KUKA KRL program: MyProgram_063().src

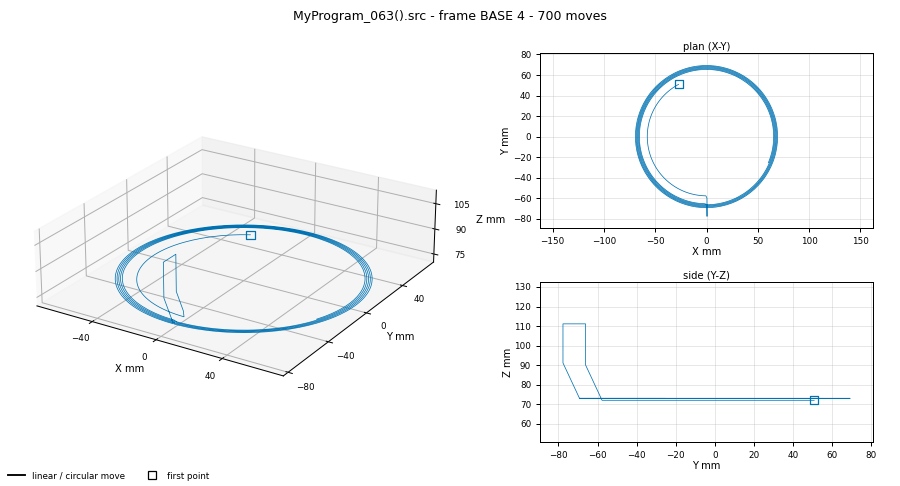
[picture p0: tool path of MyProgram_063().src in frame BASE 4, 700 of 700 moves have a stored position in this frame; points joined in program order, loops and branches not executed]
&ACCESS RVP
&REL 1
&PARAM TEMPLATE = C:\KRC\Roboter\Template\vorgabe
&PARAM EDITMASK = *
DEF MyProgram_063()
; ---- Setting reference (Base) ----
$BASE = BASE_DATA[4]

; --------------------------
; ---- Setting tool (TCP) ----
$TOOL = TOOL_DATA[3]
; --------------------------

$VEL.CP = VEL_APROX_PRINT
Startdeposition()
$VEL.CP = VEL_PRINT
LIN {X -27.2088,Y 50.891,Z 72,A 112.2891,B 24.8573,C -2.7565,E1 24.923,E2 -28.5413} C_DIS
LIN {X -29.6669,Y 49.4984,Z 72,A 115.1236,B 24.8577,C -2.7521,E1 24.9161,E2 -31.3738} C_DIS
LIN {X -32.0537,Y 47.9875,Z 72,A 117.9461,B 24.8583,C -2.7472,E1 24.9095,E2 -34.1937} C_DIS
LIN {X -34.3644,Y 46.3604,Z 72,A 120.7752,B 24.8588,C -2.742,E1 24.9031,E2 -37.0202} C_DIS
LIN {X -36.6119,Y 44.6068,Z 72,A 123.5826,B 24.8595,C -2.7356,E1 24.897,E2 -39.8228} C_DIS
LIN {X -38.7479,Y 42.7649,Z 72,A 126.4499,B 24.86,C -2.7305,E1 24.891,E2 -42.6893} C_DIS
LIN {X -40.7899,Y 40.8218,Z 72,A 129.2609,B 24.8606,C -2.7241,E1 24.8854,E2 -45.4969} C_DIS
LIN {X -42.7465,Y 38.7683,Z 72,A 132.0709,B 24.8613,C -2.7171,E1 24.8801,E2 -48.3025} C_DIS
LIN {X -44.6073,Y 36.6114,Z 72,A 134.9183,B 24.862,C -2.7103,E1 24.875,E2 -51.1466} C_DIS
LIN {X -46.3432,Y 34.3876,Z 72,A 137.7118,B 24.8628,C -2.7028,E1 24.8703,E2 -53.9356} C_DIS
LIN {X -47.9666,Y 32.0848,Z 72,A 140.5939,B 24.8634,C -2.6967,E1 24.8657,E2 -56.8174} C_DIS
LIN {X -49.5558,Y 29.5705,Z 72,A 143.4336,B 24.8645,C -2.6865,E1 24.8616,E2 -59.6473} C_DIS
LIN {X -50.8913,Y 27.2082,Z 72,A 146.2802,B 24.865,C -2.6814,E1 24.8578,E2 -62.4967} C_DIS
LIN {X -52.2094,Y 24.5834,Z 72,A 149.1598,B 24.8659,C -2.6723,E1 24.8543,E2 -65.37} C_DIS
LIN {X -53.3151,Y 22.0828,Z 72,A 151.9081,B 24.8667,C -2.6647,E1 24.8512,E2 -68.1155} C_DIS
LIN {X -54.3384,Y 19.4281,Z 72,A 154.7769,B 24.8674,C -2.657,E1 24.8485,E2 -70.9819} C_DIS
LIN {X -55.2245,Y 16.7453,Z 72,A 157.5583,B 24.8683,C -2.6479,E1 24.8461,E2 -73.7577} C_DIS
LIN {X -56.0051,Y 13.9133,Z 72,A 160.45,B 24.8693,C -2.6385,E1 24.8441,E2 -76.6436} C_DIS
LIN {X -56.5972,Y 11.2653,Z 72,A 163.2006,B 24.87,C -2.631,E1 24.8425,E2 -79.3926} C_DIS
LIN {X -57.0834,Y 8.4678,Z 72,A 166.0768,B 24.8708,C -2.6231,E1 24.8412,E2 -82.2669} C_DIS
LIN {X -57.43,Y 5.6498,Z 72,A 168.848,B 24.8718,C -2.6134,E1 24.8404,E2 -85.0315} C_DIS
LIN {X -57.638,Y 2.8318,Z 72,A 171.7312,B 24.8725,C -2.6058,E1 24.8399,E2 -87.914} C_DIS
LIN {X -57.7082,Y -0.0206,Z 72,A 174.6003,B 24.8733,C -2.5975,E1 24.8398,E2 -90.7805} C_DIS
LIN {X -57.6375,Y -2.8407,Z 72,A 177.3607,B 24.8742,C -2.588,E1 24.8401,E2 -93.5348} C_DIS
LIN {X -57.4183,Y -5.7684,Z 72,A -179.6933,B 24.8751,C -2.5795,E1 24.8408,E2 -96.478} C_DIS
LIN {X -57.0846,Y -8.4591,Z 72,A -176.9668,B 24.8758,C -2.5717,E1 24.8418,E2 -99.2022} C_DIS
LIN {X -56.5987,Y -11.258,Z 72,A -174.1104,B 24.8766,C -2.5637,E1 24.8433,E2 -102.0565} C_DIS
LIN {X -55.9773,Y -14.0247,Z 72,A -171.2895,B 24.8774,C -2.5553,E1 24.8451,E2 -104.8738} C_DIS
LIN {X -55.2229,Y -16.7506,Z 72,A -168.4174,B 24.8781,C -2.548,E1 24.8473,E2 -107.7451} C_DIS
LIN {X -54.3355,Y -19.4363,Z 72,A -165.6279,B 24.8789,C -2.5396,E1 24.8499,E2 -110.5302} C_DIS
LIN {X -53.3047,Y -22.108,Z 72,A -162.771,B 24.8797,C -2.5317,E1 24.8528,E2 -113.3843} C_DIS
LIN {X -52.1127,Y -24.7874,Z 72,A -159.8924,B 24.8805,C -2.523,E1 24.8562,E2 -116.2579} C_DIS
LIN {X -50.8921,Y -27.2066,Z 72,A -157.1453,B 24.8811,C -2.5168,E1 24.8597,E2 -119.0047} C_DIS
LIN {X -49.5012,Y -29.6623,Z 72,A -154.3076,B 24.8817,C -2.51,E1 24.8637,E2 -121.8411} C_DIS
LIN {X -47.9927,Y -32.0459,Z 72,A -151.4699,B 24.8823,C -2.5036,E1 24.868,E2 -124.6778} C_DIS
LIN {X -46.3598,Y -34.3651,Z 72,A -148.6733,B 24.883,C -2.4965,E1 24.8726,E2 -127.4709} C_DIS
LIN {X -44.6722,Y -36.5319,Z 72,A -145.9581,B 24.8836,C -2.4899,E1 24.8773,E2 -130.1831} C_DIS
LIN {X -42.9715,Y -38.5173,Z 72,A -143.3305,B 24.8841,C -2.4847,E1 24.8822,E2 -132.8102} C_DIS
LIN {X -41.017,Y -40.5923,Z 72,A -140.4968,B 24.8847,C -2.4788,E1 24.8877,E2 -135.642} C_DIS
LIN {X -38.9797,Y -42.5525,Z 72,A -137.6509,B 24.8851,C -2.4739,E1 24.8935,E2 -138.4878} C_DIS
LIN {X -36.8321,Y -44.4244,Z 72,A -134.8917,B 24.8857,C -2.4673,E1 24.8993,E2 -141.2419} C_DIS
LIN {X -34.7623,Y -46.0622,Z 72,A -132.2373,B 24.8861,C -2.4633,E1 24.9052,E2 -143.8966} C_DIS
LIN {X -32.6406,Y -47.5903,Z 72,A -129.5668,B 24.8864,C -2.4605,E1 24.9113,E2 -146.5694} C_DIS
LIN {X -30.2771,Y -49.1274,Z 72,A -126.7787,B 24.8868,C -2.4561,E1 24.9179,E2 -149.356} C_DIS
LIN {X -27.8422,Y -50.5472,Z 72,A -123.9046,B 24.887,C -2.4537,E1 24.9249,E2 -152.2328} C_DIS
LIN {X -25.3395,Y -51.8463,Z 72,A -121.1321,B 24.8874,C -2.4498,E1 24.9318,E2 -155.0034} C_DIS
LIN {X -22.7304,Y -53.0422,Z 72,A -118.294,B 24.8877,C -2.4465,E1 24.939,E2 -157.8405} C_DIS
LIN {X -19.9996,Y -54.1309,Z 72,A -115.4113,B 24.888,C -2.4431,E1 24.9465,E2 -160.7212} C_DIS
LIN {X -17.431,Y -55.0116,Z 72,A -112.6658,B 24.888,C -2.442,E1 24.9538,E2 -163.4692} C_DIS
LIN {X -14.707,Y -55.8019,Z 72,A -109.8374,B 24.8882,C -2.4405,E1 24.9614,E2 -166.2983} C_DIS
LIN {X -11.8501,Y -56.478,Z 72,A -106.9721,B 24.8884,C -2.4382,E1 24.9692,E2 -169.1617} C_DIS
LIN {X -9.1675,Y -56.9755,Z 72,A -104.197,B 24.8884,C -2.4386,E1 24.9769,E2 -171.9406} C_DIS
LIN {X -6.3785,Y -57.3539,Z 72,A -101.389,B 24.8884,C -2.4385,E1 24.9847,E2 -174.7502} C_DIS
LIN {X -3.4748,Y -57.6033,Z 72,A -98.5125,B 24.8884,C -2.4381,E1 24.9927,E2 -177.627} C_DIS
LIN {X -0.6243,Y -57.7045,Z 72,A -95.7298,B 24.8884,C -2.4375,E1 25.0004,E2 -180.4086} C_DIS
LIN {X -0.6243,Y -57.7045,Z 72,A -95.7298,B 24.8884,C -2.4375,E1 25.0004,E2 -180.4086} C_DIS
Enddeposition()
LIN {X 0.4164,Y -59.8168,Z 76.5315,A -95.6722,B 24.8907,C -2.4133,E1 25.0004,E2 -180.4086} C_DIS
LIN {X 0.4214,Y -66.1561,Z 90.1262,A -95.6453,B 24.8917,C -2.402,E1 25.0004,E2 -180.4086} C_DIS
LIN {X 0.4214,Y -66.1561,Z 111.1262,A -96.001,B 24.8778,C -2.5516,E1 25.0004,E2 -180.4086} C_DIS
LIN {X 0.5054,Y -77.7039,Z 111.1262,A -95.259,B 24.8948,C -2.368,E1 25.0013,E2 -180.7142} C_DIS
LIN {X 0.5054,Y -77.7039,Z 91.1262,A -94.9205,B 24.9071,C -2.2255,E1 25.0013,E2 -180.7142} C_DIS
LIN {X 0.4665,Y -71.3647,Z 77.5315,A -94.9453,B 24.9062,C -2.2359,E1 25.0013,E2 -180.7142} C_DIS
LIN {X 0.4536,Y -69.2517,Z 73,A -94.9551,B 24.9059,C -2.2401,E1 25.0013,E2 -180.7142} C_DIS
Startdeposition()
$VEL.CP = VEL_PRINT
LIN {X -1.6996,Y -69.2353,Z 73,A -97.3478,B 24.9072,C -2.2246,E1 24.9945,E2 -178.2848} C_DIS
LIN {X -4.2468,Y -69.1258,Z 73,A -99.457,B 24.9072,C -2.2246,E1 24.9886,E2 -176.1746} C_DIS
LIN {X -6.7883,Y -68.9227,Z 73,A -101.3578,B 24.9067,C -2.2297,E1 24.9834,E2 -174.2852} C_DIS
LIN {X -9.3205,Y -68.6261,Z 73,A -103.6767,B 24.9071,C -2.225,E1 24.9769,E2 -171.9535} C_DIS
LIN {X -11.9777,Y -68.2118,Z 73,A -105.8535,B 24.907,C -2.2268,E1 24.9709,E2 -169.7789} C_DIS
LIN {X -15.0376,Y -67.6032,Z 73,A -108.2937,B 24.9066,C -2.2313,E1 24.9643,E2 -167.3464} C_DIS
LIN {X -17.651,Y -66.9691,Z 73,A -110.7147,B 24.9069,C -2.2278,E1 24.9577,E2 -164.9138} C_DIS
LIN {X -20.104,Y -66.274,Z 73,A -112.8273,B 24.9068,C -2.2292,E1 24.952,E2 -162.8009} C_DIS
LIN {X -22.5297,Y -65.4891,Z 73,A -114.914,B 24.9066,C -2.2314,E1 24.9465,E2 -160.7155} C_DIS
LIN {X -24.9249,Y -64.6155,Z 73,A -116.8452,B 24.9061,C -2.2374,E1 24.9415,E2 -158.7948} C_DIS
LIN {X -27.2864,Y -63.6543,Z 73,A -119.1684,B 24.9063,C -2.2346,E1 24.9355,E2 -156.4595} C_DIS
LIN {X -29.6108,Y -62.6068,Z 73,A -121.2832,B 24.9061,C -2.2368,E1 24.9301,E2 -154.3447} C_DIS
LIN {X -31.8951,Y -61.4745,Z 73,A -123.3985,B 24.9059,C -2.2393,E1 24.9249,E2 -152.2297} C_DIS
LIN {X -34.2574,Y -60.1892,Z 73,A -125.5804,B 24.9056,C -2.2433,E1 24.9195,E2 -150.051} C_DIS
LIN {X -36.9333,Y -58.5854,Z 73,A -127.9318,B 24.9048,C -2.2523,E1 24.914,E2 -147.7136} C_DIS
LIN {X -38.5924,Y -57.506,Z 73,A -129.8132,B 24.9051,C -2.2493,E1 24.9096,E2 -145.819} C_DIS
LIN {X -41.1431,Y -55.7096,Z 73,A -132.1658,B 24.9043,C -2.2588,E1 24.9043,E2 -143.4807} C_DIS
LIN {X -43.1657,Y -54.1575,Z 73,A -134.2837,B 24.904,C -2.2623,E1 24.8996,E2 -141.3635} C_DIS
LIN {X -45.0032,Y -52.6399,Z 73,A -136.5418,B 24.9042,C -2.2596,E1 24.8947,E2 -139.0901} C_DIS
LIN {X -47.2376,Y -50.6451,Z 73,A -138.9913,B 24.9037,C -2.2651,E1 24.8897,E2 -136.6439} C_DIS
LIN {X -49.4705,Y -48.4663,Z 73,A -141.3461,B 24.9029,C -2.2754,E1 24.885,E2 -134.3039} C_DIS
LIN {X -51.2209,Y -46.6126,Z 73,A -143.5601,B 24.9027,C -2.2777,E1 24.8808,E2 -132.0856} C_DIS
LIN {X -52.9925,Y -44.5893,Z 73,A -145.9907,B 24.9027,C -2.2782,E1 24.8764,E2 -129.6451} C_DIS
LIN {X -54.5978,Y -42.6086,Z 73,A -148.0451,B 24.9021,C -2.2843,E1 24.8728,E2 -127.5957} C_DIS
LIN {X -56.2103,Y -40.4563,Z 73,A -150.2985,B 24.9017,C -2.2891,E1 24.8691,E2 -125.3428} C_DIS
LIN {X -57.9753,Y -37.8838,Z 73,A -152.6554,B 24.9007,C -2.3004,E1 24.8655,E2 -123.0012} C_DIS
LIN {X -59.2789,Y -35.8089,Z 73,A -154.7202,B 24.9003,C -2.3048,E1 24.8624,E2 -120.9363} C_DIS
LIN {X -60.327,Y -34.0142,Z 73,A -156.6632,B 24.9003,C -2.3046,E1 24.8597,E2 -118.9825} C_DIS
LIN {X -61.7977,Y -31.2628,Z 73,A -159.0212,B 24.8993,C -2.3163,E1 24.8567,E2 -116.64} C_DIS
LIN {X -62.883,Y -29.0176,Z 73,A -161.2043,B 24.8991,C -2.3195,E1 24.8541,E2 -114.4526} C_DIS
LIN {X -63.9843,Y -26.5032,Z 73,A -163.6722,B 24.8989,C -2.3217,E1 24.8513,E2 -111.9764} C_DIS
LIN {X -64.9644,Y -23.9988,Z 73,A -165.8612,B 24.8982,C -2.3289,E1 24.8492,E2 -109.7922} C_DIS
LIN {X -65.8037,Y -21.5914,Z 73,A -167.985,B 24.8977,C -2.3347,E1 24.8473,E2 -107.6703} C_DIS
LIN {X -66.5538,Y -19.1547,Z 73,A -170.1085,B 24.8972,C -2.3407,E1 24.8456,E2 -105.5487} C_DIS
LIN {X -67.3489,Y -16.138,Z 73,A -172.468,B 24.8961,C -2.3531,E1 24.844,E2 -103.2052} C_DIS
LIN {X -67.8973,Y -13.6481,Z 73,A -174.592,B 24.8956,C -2.3593,E1 24.8427,E2 -101.0833} C_DIS
LIN {X -68.3252,Y -11.31,Z 73,A -176.8369,B 24.8956,C -2.3595,E1 24.8417,E2 -98.8256} C_DIS
LIN {X -68.7353,Y -8.4777,Z 73,A -179.0356,B 24.8946,C -2.3704,E1 24.8408,E2 -96.6397} C_DIS
LIN {X -69.0008,Y -5.942,Z 73,A 178.6296,B 24.8944,C -2.3722,E1 24.8402,E2 -94.2955} C_DIS
LIN {X -69.1727,Y -3.3982,Z 73,A 176.5051,B 24.8938,C -2.3786,E1 24.8399,E2 -92.1733} C_DIS
LIN {X -69.2526,Y -0.6533,Z 73,A 174.2028,B 24.8932,C -2.3851,E1 24.8398,E2 -89.8728} C_DIS
LIN {X -69.2092,Y 2.5491,Z 73,A 171.5482,B 24.8925,C -2.3934,E1 24.84,E2 -87.222} C_DIS
LIN {X -69.0685,Y 5.0948,Z 73,A 169.6341,B 24.8915,C -2.4041,E1 24.8403,E2 -85.3221} C_DIS
LIN {X -68.8342,Y 7.6336,Z 73,A 167.2992,B 24.8914,C -2.4061,E1 24.841,E2 -82.9779} C_DIS
LIN {X -68.5066,Y 10.162,Z 73,A 165.1746,B 24.8908,C -2.4125,E1 24.8418,E2 -80.8558} C_DIS
LIN {X -67.9862,Y 13.1957,Z 73,A 162.8452,B 24.8896,C -2.425,E1 24.8429,E2 -78.5425} C_DIS
LIN {X -67.5419,Y 15.3103,Z 73,A 160.862,B 24.8895,C -2.4266,E1 24.8441,E2 -76.5513} C_DIS
LIN {X -66.9326,Y 17.7859,Z 73,A 158.7356,B 24.8889,C -2.4328,E1 24.8456,E2 -74.4273} C_DIS
LIN {X -66.0637,Y 20.7823,Z 73,A 156.3753,B 24.8878,C -2.4453,E1 24.8475,E2 -72.0835} C_DIS
LIN {X -65.254,Y 23.1998,Z 73,A 154.1569,B 24.8874,C -2.4495,E1 24.8495,E2 -69.8625} C_DIS
LIN {X -64.3048,Y 25.716,Z 73,A 151.7219,B 24.8872,C -2.4518,E1 24.852,E2 -67.4193} C_DIS
LIN {X -63.3146,Y 28.0655,Z 73,A 149.8086,B 24.8862,C -2.4622,E1 24.8541,E2 -65.5202} C_DIS
LIN {X -62.2387,Y 30.3769,Z 73,A 147.685,B 24.8857,C -2.4681,E1 24.8566,E2 -63.3993} C_DIS
LIN {X -61.0785,Y 32.6471,Z 73,A 145.3517,B 24.8855,C -2.4695,E1 24.8597,E2 -61.0568} C_DIS
LIN {X -59.8354,Y 34.8731,Z 73,A 143.4389,B 24.8846,C -2.4797,E1 24.8623,E2 -59.1583} C_DIS
LIN {X -58.5113,Y 37.0519,Z 73,A 141.106,B 24.8845,C -2.4808,E1 24.8657,E2 -56.8163} C_DIS
LIN {X -57.1079,Y 39.1804,Z 73,A 139.0516,B 24.8838,C -2.4878,E1 24.8689,E2 -54.7682} C_DIS
LIN {X -55.6271,Y 41.2558,Z 73,A 136.8615,B 24.8835,C -2.4917,E1 24.8725,E2 -52.5768} C_DIS
LIN {X -53.9829,Y 43.3839,Z 73,A 134.6734,B 24.8828,C -2.4983,E1 24.8763,E2 -50.3942} C_DIS
LIN {X -51.9742,Y 45.7711,Z 73,A 132.222,B 24.882,C -2.5076,E1 24.8807,E2 -47.9538} C_DIS
LIN {X -50.1586,Y 47.7549,Z 73,A 130.0004,B 24.8815,C -2.5131,E1 24.885,E2 -45.7355} C_DIS
LIN {X -48.3669,Y 49.5688,Z 73,A 127.6695,B 24.8815,C -2.5133,E1 24.8896,E2 -43.3954} C_DIS
LIN {X -46.5096,Y 51.3154,Z 73,A 125.5493,B 24.881,C -2.5179,E1 24.894,E2 -41.2775} C_DIS
LIN {X -44.4818,Y 53.0819,Z 73,A 123.3632,B 24.8805,C -2.5236,E1 24.8986,E2 -39.0966} C_DIS
LIN {X -42.0461,Y 55.0313,Z 73,A 121.0085,B 24.8795,C -2.534,E1 24.9037,E2 -36.758} C_DIS
LIN {X -39.992,Y 56.5416,Z 73,A 118.8893,B 24.8791,C -2.538,E1 24.9085,E2 -34.641} C_DIS
LIN {X -37.8838,Y 57.9753,Z 73,A 116.6766,B 24.8789,C -2.5398,E1 24.9136,E2 -32.4252} C_DIS
LIN {X -35.6048,Y 59.403,Z 73,A 114.2482,B 24.8789,C -2.5394,E1 24.9194,E2 -29.9882} C_DIS
LIN {X -33.3942,Y 60.6732,Z 73,A 112.3403,B 24.8782,C -2.5474,E1 24.9241,E2 -28.094} C_DIS
LIN {X -31.1384,Y 61.8613,Z 73,A 110.0136,B 24.8783,C -2.546,E1 24.9299,E2 -25.7576} C_DIS
LIN {X -28.7129,Y 63.0229,Z 73,A 107.8309,B 24.8779,C -2.5503,E1 24.9354,E2 -23.5797} C_DIS
LIN {X -25.8454,Y 64.2521,Z 73,A 105.3814,B 24.8773,C -2.5569,E1 24.9417,E2 -21.1403} C_DIS
LIN {X -23.3317,Y 65.2077,Z 73,A 102.9603,B 24.8774,C -2.5553,E1 24.948,E2 -18.7105} C_DIS
LIN {X -20.7823,Y 66.0637,Z 73,A 100.7794,B 24.8771,C -2.5589,E1 24.9538,E2 -16.5341} C_DIS
LIN {X -17.7859,Y 66.9326,Z 73,A 98.2119,B 24.8768,C -2.5619,E1 24.9607,E2 -13.9697} C_DIS
LIN {X -15.0376,Y 67.6032,Z 73,A 95.8468,B 24.8766,C -2.5634,E1 24.9671,E2 -11.6051} C_DIS
LIN {X -11.9777,Y 68.2118,Z 73,A 93.2608,B 24.8765,C -2.5653,E1 24.9742,E2 -9.0209} C_DIS
LIN {X -9.1819,Y 68.6441,Z 73,A 90.9169,B 24.8763,C -2.5667,E1 24.9807,E2 -6.6784} C_DIS
LIN {X -6.0812,Y 68.9879,Z 73,A 88.5704,B 24.8757,C -2.5736,E1 24.9872,E2 -4.3469} C_DIS
LIN {X -4.1073,Y 69.1335,Z 73,A 86.6937,B 24.8761,C -2.5686,E1 24.9924,E2 -2.4576} C_DIS
LIN {X -0.9896,Y 69.2484,Z 73,A 84.2546,B 24.8757,C -2.5727,E1 24.9992,E2 -0.028} C_DIS
LIN {X 1.6996,Y 69.2353,Z 73,A 81.8355,B 24.8762,C -2.5684,E1 25.006,E2 2.401} C_DIS
LIN {X 4.2468,Y 69.1258,Z 73,A 79.7364,B 24.8762,C -2.5687,E1 25.0119,E2 4.4987} C_DIS
LIN {X 6.7883,Y 68.9227,Z 73,A 77.8259,B 24.8757,C -2.5733,E1 25.0171,E2 6.3972} C_DIS
LIN {X 9.3205,Y 68.6261,Z 73,A 75.5089,B 24.8762,C -2.5678,E1 25.0236,E2 8.7254} C_DIS
LIN {X 11.8402,Y 68.2365,Z 73,A 73.4007,B 24.8762,C -2.5671,E1 25.0294,E2 10.8329} C_DIS
LIN {X 14.3437,Y 67.7545,Z 73,A 71.5022,B 24.8759,C -2.5714,E1 25.0346,E2 12.7191} C_DIS
LIN {X 16.8279,Y 67.1806,Z 73,A 69.3955,B 24.8759,C -2.5703,E1 25.0403,E2 14.8254} C_DIS
LIN {X 19.2892,Y 66.5157,Z 73,A 67.0806,B 24.8766,C -2.5638,E1 25.0465,E2 17.1519} C_DIS
LIN {X 21.8568,Y 65.716,Z 73,A 64.9092,B 24.8766,C -2.5634,E1 25.0523,E2 19.3202} C_DIS
LIN {X 24.7942,Y 64.665,Z 73,A 62.5704,B 24.8763,C -2.5671,E1 25.0584,E2 21.6453} C_DIS
LIN {X 26.632,Y 63.9301,Z 73,A 60.6996,B 24.877,C -2.5596,E1 25.0633,E2 23.5296} C_DIS
LIN {X 29.4841,Y 62.6658,Z 73,A 58.3618,B 24.8767,C -2.5628,E1 25.0692,E2 25.8539} C_DIS
LIN {X 31.7707,Y 61.5381,Z 73,A 56.1647,B 24.8772,C -2.5579,E1 25.0747,E2 28.0566} C_DIS
LIN {X 34.1362,Y 60.2589,Z 73,A 53.962,B 24.8774,C -2.5555,E1 25.08,E2 30.2587} C_DIS
LIN {X 36.3311,Y 58.9616,Z 73,A 51.6513,B 24.8782,C -2.5472,E1 25.0856,E2 32.5817} C_DIS
LIN {X 38.4767,Y 57.5844,Z 73,A 49.797,B 24.8779,C -2.5505,E1 25.0899,E2 34.4223} C_DIS
LIN {X 40.5701,Y 56.1291,Z 73,A 47.4764,B 24.8787,C -2.5415,E1 25.0952,E2 36.756} C_DIS
LIN {X 42.6086,Y 54.5978,Z 73,A 45.3469,B 24.8792,C -2.5372,E1 25.0999,E2 38.8879} C_DIS
LIN {X 44.6957,Y 52.9019,Z 73,A 43.1809,B 24.8794,C -2.5346,E1 25.1046,E2 41.0518} C_DIS
LIN {X 47.0328,Y 50.8353,Z 73,A 40.8475,B 24.8793,C -2.536,E1 25.1094,E2 43.3725} C_DIS
LIN {X 48.4663,Y 49.4705,Z 73,A 38.9811,B 24.8802,C -2.5266,E1 25.1132,E2 45.2533} C_DIS
LIN {X 50.6451,Y 47.2376,Z 73,A 36.6485,B 24.8801,C -2.5276,E1 25.1177,E2 47.5735} C_DIS
LIN {X 52.3494,Y 45.3415,Z 73,A 34.4563,B 24.8807,C -2.5207,E1 25.1217,E2 49.7722} C_DIS
LIN {X 54.0709,Y 43.2754,Z 73,A 32.0505,B 24.8817,C -2.5108,E1 25.126,E2 52.1904} C_DIS
LIN {X 55.6271,Y 41.2558,Z 73,A 29.9525,B 24.8821,C -2.506,E1 25.1295,E2 54.2898} C_DIS
LIN {X 57.1079,Y 39.1804,Z 73,A 28.0625,B 24.8821,C -2.5066,E1 25.1325,E2 56.1691} C_DIS
LIN {X 58.5113,Y 37.0519,Z 73,A 25.7574,B 24.8831,C -2.496,E1 25.1361,E2 58.4877} C_DIS
LIN {X 59.9051,Y 34.752,Z 73,A 23.5949,B 24.8835,C -2.4918,E1 25.1391,E2 60.6489} C_DIS
LIN {X 61.1436,Y 32.5235,Z 73,A 21.4983,B 24.884,C -2.4865,E1 25.1419,E2 62.7471} C_DIS
LIN {X 62.5463,Y 29.7368,Z 73,A 19.1689,B 24.884,C -2.4862,E1 25.1448,E2 65.0648} C_DIS
LIN {X 63.5984,Y 27.4145,Z 73,A 17.0727,B 24.8845,C -2.4806,E1 25.1472,E2 67.1627} C_DIS
LIN {X 64.5644,Y 25.055,Z 73,A 14.8837,B 24.8853,C -2.4724,E1 25.1494,E2 69.359} C_DIS
LIN {X 65.4891,Y 22.5297,Z 73,A 12.6887,B 24.8858,C -2.4667,E1 25.1515,E2 71.5551} C_DIS
LIN {X 66.274,Y 20.104,Z 73,A 10.5932,B 24.8863,C -2.4609,E1 25.1533,E2 73.6526} C_DIS
LIN {X 66.9691,Y 17.651,Z 73,A 8.2903,B 24.8874,C -2.4492,E1 25.155,E2 75.9697} C_DIS
LIN {X 67.6032,Y 15.0376,Z 73,A 6.13,B 24.8879,C -2.4443,E1 25.1563,E2 78.1293} C_DIS
LIN {X 68.2118,Y 11.9777,Z 73,A 3.8022,B 24.8879,C -2.4433,E1 25.1575,E2 80.4458} C_DIS
LIN {X 68.5262,Y 10.0236,Z 73,A 1.9402,B 24.889,C -2.432,E1 25.1583,E2 82.3234} C_DIS
LIN {X 68.8487,Y 7.4946,Z 73,A -0.1544,B 24.8896,C -2.4258,E1 25.159,E2 84.4202} C_DIS
LIN {X 69.1164,Y 4.3863,Z 73,A -2.4819,B 24.8896,C -2.4247,E1 25.1595,E2 86.7366} C_DIS
LIN {X 69.231,Y 1.8393,Z 73,A -4.6824,B 24.8905,C -2.4155,E1 25.1598,E2 88.9458} C_DIS
LIN {X 69.2484,Y -0.9896,Z 73,A -7.1363,B 24.8915,C -2.405,E1 25.1598,E2 91.4099} C_DIS
LIN {X 69.1335,Y -4.1073,Z 73,A -9.4637,B 24.8915,C -2.4038,E1 25.1594,E2 93.7263} C_DIS
LIN {X 68.9879,Y -6.0812,Z 73,A -11.3251,B 24.8926,C -2.3924,E1 25.159,E2 95.6035} C_DIS
LIN {X 68.6441,Y -9.1819,Z 73,A -13.6521,B 24.8927,C -2.3912,E1 25.1582,E2 97.9197} C_DIS
LIN {X 68.2596,Y -11.7023,Z 73,A -15.7466,B 24.8933,C -2.3849,E1 25.1573,E2 100.0167} C_DIS
LIN {X 67.8973,Y -13.6481,Z 73,A -17.6085,B 24.8943,C -2.3736,E1 25.1563,E2 101.8945} C_DIS
LIN {X 67.2482,Y -16.551,Z 73,A -19.9474,B 24.8947,C -2.3692,E1 25.1548,E2 104.2302} C_DIS
LIN {X 66.5157,Y -19.2892,Z 73,A -22.4306,B 24.8957,C -2.3581,E1 25.153,E2 106.7253} C_DIS
LIN {X 65.716,Y -21.8568,Z 73,A -24.5909,B 24.8961,C -2.353,E1 25.1511,E2 108.8854} C_DIS
LIN {X 64.6438,Y -24.8503,Z 73,A -27.0517,B 24.8964,C -2.3497,E1 25.1487,E2 111.3404} C_DIS
LIN {X 63.6543,Y -27.2864,Z 73,A -29.4049,B 24.8974,C -2.3382,E1 25.1462,E2 113.7076} C_DIS
LIN {X 62.6068,Y -29.6108,Z 73,A -31.5095,B 24.898,C -2.3321,E1 25.1437,E2 115.8153} C_DIS
LIN {X 61.4745,Y -31.8951,Z 73,A -33.605,B 24.8985,C -2.3263,E1 25.1411,E2 117.9135} C_DIS
LIN {X 60.1892,Y -34.2574,Z 73,A -35.7664,B 24.8989,C -2.3216,E1 25.1381,E2 120.0746} C_DIS
LIN {X 58.5854,Y -36.9333,Z 73,A -38.0955,B 24.8989,C -2.3212,E1 25.1347,E2 122.3928} C_DIS
LIN {X 57.506,Y -38.5924,Z 73,A -39.9586,B 24.8998,C -2.3106,E1 25.1318,E2 124.2719} C_DIS
LIN {X 55.7096,Y -41.1431,Z 73,A -42.3817,B 24.9001,C -2.3078,E1 25.1279,E2 126.6896} C_DIS
LIN {X 54.0709,Y -43.2754,Z 73,A -44.7858,B 24.901,C -2.2971,E1 25.1237,E2 129.1077} C_DIS
LIN {X 52.4414,Y -45.2362,Z 73,A -46.8829,B 24.9014,C -2.2921,E1 25.1199,E2 131.2073} C_DIS
LIN {X 50.6451,Y -47.2376,Z 73,A -49.0462,B 24.9018,C -2.2882,E1 25.1159,E2 133.3702} C_DIS
LIN {X 48.4663,Y -49.4705,Z 73,A -51.3776,B 24.9018,C -2.2887,E1 25.1113,E2 135.6905} C_DIS
LIN {X 46.6126,Y -51.2209,Z 73,A -53.5693,B 24.9023,C -2.2815,E1 25.1068,E2 137.8901} C_DIS
LIN {X 44.5893,Y -52.9925,Z 73,A -55.9754,B 24.9032,C -2.2717,E1 25.1017,E2 140.31} C_DIS
LIN {X 42.6086,Y -54.5978,Z 73,A -57.8668,B 24.9031,C -2.273,E1 25.0976,E2 142.1915} C_DIS
LIN {X 40.5701,Y -56.1291,Z 73,A -59.9665,B 24.9034,C -2.2689,E1 25.0928,E2 144.2934} C_DIS
LIN {X 38.4767,Y -57.5844,Z 73,A -62.2743,B 24.9042,C -2.2595,E1 25.0875,E2 146.6156} C_DIS
LIN {X 36.2647,Y -59.0019,Z 73,A -64.4239,B 24.9045,C -2.256,E1 25.0824,E2 148.7665} C_DIS
LIN {X 34.0142,Y -60.327,Z 73,A -66.5416,B 24.9047,C -2.2533,E1 25.0773,E2 150.8842} C_DIS
LIN {X 31.2628,Y -61.7977,Z 73,A -68.8766,B 24.9046,C -2.2554,E1 25.0715,E2 153.2077} C_DIS
LIN {X 28.967,Y -62.9065,Z 73,A -71.0722,B 24.905,C -2.2499,E1 25.066,E2 155.4107} C_DIS
LIN {X 26.5032,Y -63.9843,Z 73,A -73.4825,B 24.9057,C -2.2418,E1 25.0597,E2 157.8344} C_DIS
LIN {X 23.9988,Y -64.9644,Z 73,A -75.6514,B 24.9058,C -2.2403,E1 25.0541,E2 160.0023} C_DIS
LIN {X 21.5914,Y -65.8037,Z 73,A -77.7549,B 24.9061,C -2.2379,E1 25.0485,E2 162.1075} C_DIS
LIN {X 19.1547,Y -66.5538,Z 73,A -79.859,B 24.9062,C -2.2356,E1 25.0429,E2 164.2132} C_DIS
LIN {X 16.138,Y -67.3489,Z 73,A -82.1974,B 24.9059,C -2.2392,E1 25.0366,E2 166.5395} C_DIS
LIN {X 13.7809,Y -67.8701,Z 73,A -84.2278,B 24.9062,C -2.2366,E1 25.031,E2 168.5735} C_DIS
LIN {X 11.7023,Y -68.2596,Z 73,A -86.1741,B 24.9067,C -2.2302,E1 25.0256,E2 170.5328} C_DIS
LIN {X 9.1819,Y -68.6441,Z 73,A -88.2804,B 24.9068,C -2.2289,E1 25.0198,E2 172.6405} C_DIS
LIN {X 6.0812,Y -68.9879,Z 73,A -90.6215,B 24.9064,C -2.2335,E1 25.0133,E2 174.9692} C_DIS
LIN {X 4.1073,Y -69.1335,Z 73,A -92.4945,B 24.907,C -2.2269,E1 25.0081,E2 176.857} C_DIS
LIN {X 0.9896,Y -69.2484,Z 73,A -94.9304,B 24.9067,C -2.2297,E1 25.0013,E2 179.2858} C_DIS
LIN {X 0.9896,Y -69.2484,Z 73,A -94.9304,B 24.9067,C -2.2297,E1 25.0013,E2 179.2858} C_DIS
Enddeposition()
LIN {X 0.4496,Y -68.3008,Z 73,A -95.0992,B 24.9048,C -2.253,E1 25.001,E2 179.3991} C_DIS
Startdeposition()
$VEL.CP = VEL_PRINT
LIN {X 2.363,Y -68.2646,Z 73,A -92.8977,B 24.9035,C -2.2681,E1 25.0072,E2 177.1622} C_DIS
LIN {X 4.8793,Y -68.131,Z 73,A -90.6227,B 24.9031,C -2.273,E1 25.0136,E2 174.8765} C_DIS
LIN {X 9.2654,Y -67.6745,Z 73,A -87.0265,B 24.9031,C -2.2726,E1 25.0236,E2 171.2838} C_DIS
LIN {X 11.3581,Y -67.3541,Z 73,A -85.1881,B 24.9029,C -2.2755,E1 25.0286,E2 169.4404} C_DIS
LIN {X 14.4066,Y -66.7685,Z 73,A -81.9644,B 24.9013,C -2.2936,E1 25.0376,E2 166.1779} C_DIS
LIN {X 18.8356,Y -65.657,Z 73,A -78.7736,B 24.9024,C -2.2812,E1 25.0461,E2 163.0217} C_DIS
LIN {X 21.716,Y -64.7611,Z 73,A -76.2244,B 24.9021,C -2.2847,E1 25.0528,E2 160.4689} C_DIS
LIN {X 26.2245,Y -63.071,Z 73,A -72.5514,B 24.9024,C -2.2807,E1 25.0624,E2 156.8135} C_DIS
LIN {X 29.208,Y -61.7465,Z 73,A -69.4994,B 24.9014,C -2.293,E1 25.0702,E2 153.7399} C_DIS
LIN {X 31.8558,Y -60.4217,Z 73,A -66.4474,B 24.8997,C -2.3121,E1 25.0778,E2 150.6512} C_DIS
LIN {X 35.9068,Y -58.1066,Z 73,A -63.1095,B 24.9004,C -2.3039,E1 25.0858,E2 147.3429} C_DIS
LIN {X 38.7149,Y -56.2746,Z 73,A -60.4041,B 24.9002,C -2.3065,E1 25.0921,E2 144.6403} C_DIS
LIN {X 41.5957,Y -54.1791,Z 73,A -57.0624,B 24.8988,C -2.3222,E1 25.0996,E2 141.2736} C_DIS
LIN {X 45.1085,Y -51.2917,Z 73,A -53.8719,B 24.8995,C -2.3139,E1 25.1063,E2 138.1149} C_DIS
LIN {X 46.6282,Y -49.9142,Z 73,A -51.9251,B 24.8987,C -2.324,E1 25.1104,E2 136.1522} C_DIS
LIN {X 49.1885,Y -47.3926,Z 73,A -48.4952,B 24.897,C -2.3425,E1 25.1172,E2 132.6933} C_DIS
LIN {X 52.3173,Y -43.9156,Z 73,A -45.2559,B 24.8978,C -2.3338,E1 25.1231,E2 129.4889} C_DIS
LIN {X 53.4954,Y -42.4716,Z 73,A -43.478,B 24.8969,C -2.3437,E1 25.1262,E2 127.6959} C_DIS
LIN {X 55.1376,Y -40.3164,Z 73,A -41.2234,B 24.8964,C -2.3493,E1 25.13,E2 125.4388} C_DIS
LIN {X 56.9079,Y -37.777,Z 73,A -38.0537,B 24.8944,C -2.3721,E1 25.135,E2 122.2309} C_DIS
LIN {X 59.096,Y -34.2533,Z 73,A -35.0452,B 24.8947,C -2.369,E1 25.1393,E2 119.2451} C_DIS
LIN {X 60.64,Y -31.4407,Z 73,A -32.4274,B 24.8942,C -2.3748,E1 25.1427,E2 116.6274} C_DIS
LIN {X 62.2937,Y -28.019,Z 73,A -29.567,B 24.8942,C -2.3753,E1 25.1461,E2 113.7813} C_DIS
LIN {X 63.096,Y -26.165,Z 73,A -27.5372,B 24.8928,C -2.3896,E1 25.1483,E2 111.729} C_DIS
LIN {X 64.206,Y -23.3061,Z 73,A -24.5028,B 24.891,C -2.4102,E1 25.1513,E2 108.6628} C_DIS
LIN {X 65.5762,Y -19.1165,Z 73,A -21.3142,B 24.8912,C -2.4075,E1 25.1539,E2 105.4987} C_DIS
LIN {X 66.2927,Y -16.4596,Z 73,A -19.0003,B 24.8906,C -2.4149,E1 25.1555,E2 103.1807} C_DIS
LIN {X 67.0508,Y -13.0297,Z 73,A -16.4096,B 24.8906,C -2.4143,E1 25.157,E2 100.6063} C_DIS
LIN {X 67.4272,Y -10.9209,Z 73,A -14.308,B 24.8893,C -2.4284,E1 25.158,E2 98.4838} C_DIS
LIN {X 67.8197,Y -8.1297,Z 73,A -12.058,B 24.8889,C -2.4328,E1 25.1588,E2 96.2368} C_DIS
LIN {X 68.0866,Y -5.4576,Z 73,A -9.8303,B 24.8883,C -2.4392,E1 25.1594,E2 94.007} C_DIS
LIN {X 68.2601,Y -2.5065,Z 73,A -7.2425,B 24.8873,C -2.4501,E1 25.1597,E2 91.409} C_DIS
LIN {X 68.3042,Y -0.2376,Z 73,A -5.3104,B 24.8867,C -2.4569,E1 25.1597,E2 89.4722} C_DIS
LIN {X 68.2248,Y 3.332,Z 73,A -2.3022,B 24.8858,C -2.4667,E1 25.1595,E2 86.4588} C_DIS
LIN {X 68.0181,Y 6.2537,Z 73,A -0.132,B 24.8858,C -2.4665,E1 25.159,E2 84.3018} C_DIS
LIN {X 67.7245,Y 8.8861,Z 73,A 2.2879,B 24.8847,C -2.4789,E1 25.1582,E2 81.867} C_DIS
LIN {X 67.3185,Y 11.5707,Z 73,A 4.4521,B 24.8843,C -2.4828,E1 25.1572,E2 79.7062} C_DIS
LIN {X 66.7736,Y 14.3834,Z 73,A 6.833,B 24.8837,C -2.4896,E1 25.1559,E2 77.3233} C_DIS
LIN {X 65.8883,Y 18.0094,Z 73,A 10.4208,B 24.8816,C -2.5116,E1 25.1533,E2 73.7042} C_DIS
LIN {X 64.2268,Y 23.249,Z 73,A 14.1145,B 24.8827,C -2.5001,E1 25.1501,E2 70.0586} C_DIS
LIN {X 63.051,Y 26.272,Z 73,A 16.9298,B 24.8817,C -2.5104,E1 25.1473,E2 67.2344} C_DIS
LIN {X 62.2404,Y 28.1373,Z 73,A 18.8939,B 24.8806,C -2.5222,E1 25.145,E2 65.2532} C_DIS
LIN {X 61.0409,Y 30.6546,Z 73,A 21.4612,B 24.8794,C -2.5348,E1 25.1418,E2 62.6698} C_DIS
LIN {X 58.8637,Y 34.6503,Z 73,A 25.602,B 24.8776,C -2.5537,E1 25.1361,E2 58.5057} C_DIS
LIN {X 57.0499,Y 37.5617,Z 73,A 27.8133,B 24.8786,C -2.5431,E1 25.1328,E2 56.3307} C_DIS
LIN {X 55.6311,Y 39.6326,Z 73,A 29.9109,B 24.8781,C -2.5481,E1 25.1294,E2 54.2315} C_DIS
LIN {X 54.0858,Y 41.7168,Z 73,A 32.238,B 24.8772,C -2.5573,E1 25.1255,E2 51.8937} C_DIS
LIN {X 52.1311,Y 44.1357,Z 73,A 34.7219,B 24.877,C -2.5601,E1 25.1211,E2 49.4147} C_DIS
LIN {X 50.0884,Y 46.4418,Z 73,A 37.0817,B 24.877,C -2.5598,E1 25.1167,E2 47.0659} C_DIS
LIN {X 47.769,Y 48.8242,Z 73,A 40.1454,B 24.8757,C -2.5729,E1 25.1106,E2 43.9843} C_DIS
LIN {X 45.3133,Y 51.1114,Z 73,A 43.0274,B 24.875,C -2.5803,E1 25.1047,E2 41.0966} C_DIS
LIN {X 42.7918,Y 53.24,Z 73,A 45.7025,B 24.8747,C -2.583,E1 25.0989,E2 38.4252} C_DIS
LIN {X 40.4275,Y 55.0562,Z 73,A 48.0103,B 24.8748,C -2.5824,E1 25.0938,E2 36.1272} C_DIS
LIN {X 38.6282,Y 56.3346,Z 73,A 50.3965,B 24.8732,C -2.5992,E1 25.0882,E2 33.7093} C_DIS
LIN {X 36.1165,Y 57.9756,Z 73,A 52.729,B 24.8732,C -2.5983,E1 25.0828,E2 31.3865} C_DIS
LIN {X 33.0581,Y 59.7729,Z 73,A 55.4677,B 24.8734,C -2.5964,E1 25.0761,E2 28.6604} C_DIS
LIN {X 30.7936,Y 60.9707,Z 73,A 57.5985,B 24.8732,C -2.5987,E1 25.0709,E2 26.5302} C_DIS
LIN {X 28.4739,Y 62.0882,Z 73,A 59.7647,B 24.873,C -2.6013,E1 25.0654,E2 24.3632} C_DIS
LIN {X 26.2059,Y 63.0788,Z 73,A 61.9529,B 24.8725,C -2.6064,E1 25.0597,E2 22.1682} C_DIS
LIN {X 23.0718,Y 64.2914,Z 73,A 64.5558,B 24.8727,C -2.6035,E1 25.053,E2 19.5776} C_DIS
LIN {X 19.7748,Y 65.3797,Z 73,A 67.6849,B 24.872,C -2.6112,E1 25.0446,E2 16.4361} C_DIS
LIN {X 15.4049,Y 66.5451,Z 73,A 71.355,B 24.872,C -2.6104,E1 25.0347,E2 12.7735} C_DIS
LIN {X 10.478,Y 67.4965,Z 73,A 75.5358,B 24.872,C -2.6112,E1 25.0232,E2 8.5953} C_DIS
LIN {X 7.5762,Y 67.8845,Z 73,A 78.0975,B 24.8717,C -2.6143,E1 25.0161,E2 6.0284} C_DIS
LIN {X 4.5034,Y 68.1564,Z 73,A 81.3194,B 24.8702,C -2.6297,E1 25.007,E2 2.7712} C_DIS
LIN {X 0.4169,Y 68.3037,Z 73,A 84.0772,B 24.8718,C -2.6131,E1 24.9995,E2 0.0534} C_DIS
LIN {X -3.273,Y 68.2273,Z 73,A 87.0194,B 24.8722,C -2.6085,E1 24.9913,E2 -2.8783} C_DIS
LIN {X -5.9489,Y 68.0462,Z 73,A 89.4313,B 24.872,C -2.6113,E1 24.9845,E2 -5.298} C_DIS
LIN {X -8.7582,Y 67.7411,Z 73,A 91.6776,B 24.8724,C -2.6071,E1 24.9783,E2 -7.5357} C_DIS
LIN {X -11.3284,Y 67.359,Z 73,A 94.0127,B 24.8722,C -2.6092,E1 24.9719,E2 -9.878} C_DIS
LIN {X -15.1657,Y 66.6004,Z 73,A 97.2351,B 24.8726,C -2.6051,E1 24.9631,E2 -13.0944} C_DIS
LIN {X -18.2483,Y 65.8234,Z 73,A 99.9039,B 24.8728,C -2.6025,E1 24.9559,E2 -15.761} C_DIS
LIN {X -20.8095,Y 65.0583,Z 73,A 102.1355,B 24.8731,C -2.5997,E1 24.9499,E2 -17.9899} C_DIS
LIN {X -23.3593,Y 64.1865,Z 73,A 104.3485,B 24.8735,C -2.5959,E1 24.9441,E2 -20.1981} C_DIS
LIN {X -25.9327,Y 63.191,Z 73,A 106.6687,B 24.8738,C -2.5929,E1 24.9381,E2 -22.5162} C_DIS
LIN {X -28.4842,Y 62.0835,Z 73,A 109.2309,B 24.8736,C -2.5946,E1 24.9315,E2 -25.0886} C_DIS
LIN {X -31.1275,Y 60.8001,Z 73,A 111.2639,B 24.8749,C -2.5811,E1 24.9265,E2 -27.0947} C_DIS
LIN {X -33.1356,Y 59.7297,Z 73,A 114.5866,B 24.8721,C -2.6096,E1 24.9182,E2 -30.495} C_DIS
LIN {X -36.7242,Y 57.5929,Z 73,A 116.8493,B 24.8755,C -2.5754,E1 24.9131,E2 -32.6832} C_DIS
LIN {X -38.62,Y 56.3402,Z 73,A 119.0027,B 24.8753,C -2.5771,E1 24.908,E2 -34.848} C_DIS
LIN {X -41.0843,Y 54.5678,Z 73,A 122.1676,B 24.8745,C -2.5856,E1 24.9009,E2 -38.0444} C_DIS
LIN {X -45.0912,Y 51.3069,Z 73,A 125.9063,B 24.8767,C -2.563,E1 24.893,E2 -41.7437} C_DIS
LIN {X -47.2828,Y 49.2943,Z 73,A 128.3019,B 24.8774,C -2.5551,E1 24.8881,E2 -44.1302} C_DIS
LIN {X -49.2261,Y 47.3535,Z 73,A 130.8246,B 24.8775,C -2.5543,E1 24.8832,E2 -46.6617} C_DIS
LIN {X -51.2337,Y 45.1748,Z 73,A 133.5575,B 24.8775,C -2.5534,E1 24.8781,E2 -49.4049} C_DIS
LIN {X -54.4456,Y 41.247,Z 73,A 137.3987,B 24.8795,C -2.5335,E1 24.8715,E2 -53.2164} C_DIS
LIN {X -56.6323,Y 38.1885,Z 73,A 140.9703,B 24.8795,C -2.5338,E1 24.8657,E2 -56.8065} C_DIS
LIN {X -58.2412,Y 35.6875,Z 73,A 143.124,B 24.8808,C -2.5196,E1 24.8626,E2 -58.9372} C_DIS
LIN {X -59.7245,Y 33.1448,Z 73,A 145.6468,B 24.8814,C -2.5137,E1 24.8591,E2 -61.4591} C_DIS
LIN {X -61.0608,Y 30.6144,Z 73,A 147.9794,B 24.8822,C -2.5053,E1 24.8561,E2 -63.7841} C_DIS
LIN {X -62.1493,Y 28.3394,Z 73,A 150.1516,B 24.8827,C -2.5003,E1 24.8536,E2 -65.9561} C_DIS
LIN {X -63.1948,Y 25.9232,Z 73,A 152.2592,B 24.8835,C -2.4915,E1 24.8513,E2 -68.0546} C_DIS
LIN {X -64.1022,Y 23.5905,Z 73,A 154.4012,B 24.884,C -2.4861,E1 24.8492,E2 -70.1955} C_DIS
LIN {X -64.9421,Y 21.1688,Z 73,A 156.5155,B 24.8847,C -2.4787,E1 24.8473,E2 -72.3043} C_DIS
LIN {X -65.7008,Y 18.6808,Z 73,A 158.5174,B 24.8857,C -2.4683,E1 24.8457,E2 -74.2928} C_DIS
LIN {X -66.2545,Y 16.6151,Z 73,A 160.7173,B 24.8854,C -2.4711,E1 24.8442,E2 -76.5123} C_DIS
LIN {X -67.2488,Y 11.9658,Z 73,A 164.4102,B 24.8871,C -2.4524,E1 24.8421,E2 -80.1824} C_DIS
LIN {X -67.5255,Y 10.2905,Z 73,A 166.1105,B 24.8871,C -2.4537,E1 24.8414,E2 -81.8958} C_DIS
LIN {X -67.895,Y 7.4817,Z 73,A 169.0903,B 24.8865,C -2.4588,E1 24.8404,E2 -84.9058} C_DIS
LIN {X -68.2694,Y 2.2064,Z 73,A 172.7982,B 24.8892,C -2.4295,E1 24.8398,E2 -88.5658} C_DIS
LIN {X -68.2966,Y -1.0833,Z 73,A 176.0575,B 24.8891,C -2.4312,E1 24.8398,E2 -91.8489} C_DIS
LIN {X -68.1708,Y -4.2905,Z 73,A 179.3401,B 24.8887,C -2.4353,E1 24.8404,E2 -95.1609} C_DIS
LIN {X -67.8526,Y -7.8485,Z 73,A -179.0013,B 24.8921,C -2.3977,E1 24.8409,E2 -96.7396} C_DIS
LIN {X -67.3597,Y -11.3245,Z 73,A -175.6613,B 24.8921,C -2.3968,E1 24.8423,E2 -100.0974} C_DIS
LIN {X -66.9301,Y -13.6357,Z 73,A -173.7773,B 24.8929,C -2.3889,E1 24.8432,E2 -101.9738} C_DIS
LIN {X -66.4194,Y -15.9403,Z 73,A -171.5902,B 24.8931,C -2.3873,E1 24.8446,E2 -104.1697} C_DIS
LIN {X -65.6949,Y -18.7016,Z 73,A -169.1279,B 24.8936,C -2.3815,E1 24.8464,E2 -106.6326} C_DIS
LIN {X -64.8116,Y -21.5661,Z 73,A -166.6384,B 24.8943,C -2.3736,E1 24.8486,E2 -109.1174} C_DIS
LIN {X -63.5859,Y -24.9478,Z 73,A -163.7499,B 24.8953,C -2.3621,E1 24.8514,E2 -111.9949} C_DIS
LIN {X -62.5954,Y -27.3383,Z 73,A -161.408,B 24.8955,C -2.3597,E1 24.8539,E2 -114.3438} C_DIS
LIN {X -61.3751,Y -29.9803,Z 73,A -158.8894,B 24.896,C -2.3546,E1 24.8569,E2 -116.8639} C_DIS
LIN {X -59.4535,Y -33.6302,Z 73,A -155.347,B 24.8966,C -2.3471,E1 24.8617,E2 -120.4071} C_DIS
LIN {X -57.6435,Y -36.6453,Z 73,A -151.9853,B 24.8966,C -2.3485,E1 24.8667,E2 -123.7893} C_DIS
LIN {X -54.3508,Y -41.3729,Z 73,A -147.2534,B 24.8977,C -2.3345,E1 24.8744,E2 -128.5108} C_DIS
LIN {X -51.9746,Y -44.3193,Z 73,A -144.3931,B 24.899,C -2.3202,E1 24.8795,E2 -131.3503} C_DIS
LIN {X -49.9105,Y -46.6321,Z 73,A -141.7899,B 24.8995,C -2.3146,E1 24.8844,E2 -133.9516} C_DIS
LIN {X -47.3153,Y -49.263,Z 73,A -138.356,B 24.8994,C -2.3157,E1 24.8912,E2 -137.4024} C_DIS
LIN {X -44.8759,Y -51.4949,Z 73,A -135.8844,B 24.9004,C -2.3035,E1 24.8963,E2 -139.8549} C_DIS
LIN {X -40.6378,Y -54.9023,Z 73,A -131.2967,B 24.9011,C -2.296,E1 24.9064,E2 -144.4415} C_DIS
LIN {X -37.9609,Y -56.7864,Z 73,A -128.3294,B 24.9011,C -2.2966,E1 24.9133,E2 -147.4204} C_DIS
LIN {X -35.7292,Y -58.2158,Z 73,A -126.3769,B 24.9019,C -2.2871,E1 24.9179,E2 -149.3563} C_DIS
LIN {X -33.0903,Y -59.755,Z 73,A -123.8941,B 24.9023,C -2.2818,E1 24.9239,E2 -151.8338} C_DIS
LIN {X -30.9424,Y -60.8947,Z 73,A -121.648,B 24.9021,C -2.284,E1 24.9295,E2 -154.0913} C_DIS
LIN {X -27.9619,Y -62.3194,Z 73,A -118.8292,B 24.9023,C -2.282,E1 24.9366,E2 -156.9123} C_DIS
LIN {X -25.0925,Y -63.5291,Z 73,A -115.294,B 24.9006,C -2.3013,E1 24.946,E2 -160.5012} C_DIS
LIN {X -21.2472,Y -64.9167,Z 73,A -113.1188,B 24.9034,C -2.2688,E1 24.9515,E2 -162.603} C_DIS
LIN {X -19.5682,Y -65.4421,Z 73,A -111.524,B 24.9033,C -2.2705,E1 24.9558,E2 -164.2048} C_DIS
LIN {X -16.8519,Y -66.1937,Z 73,A -108.5442,B 24.9021,C -2.2839,E1 24.9639,E2 -167.2207} C_DIS
LIN {X -12.5403,Y -67.145,Z 73,A -105.2624,B 24.9031,C -2.2722,E1 24.9728,E2 -170.4785} C_DIS
LIN {X -9.3779,Y -67.6585,Z 73,A -102.6882,B 24.9034,C -2.2688,E1 24.9799,E2 -173.0469} C_DIS
LIN {X -6.8026,Y -67.9661,Z 73,A -100.1863,B 24.9028,C -2.2765,E1 24.9869,E2 -175.5686} C_DIS
LIN {X -3.551,Y -68.2129,Z 73,A -97.7514,B 24.9034,C -2.2692,E1 24.9937,E2 -177.987} C_DIS
LIN {X -0.3434,Y -68.3041,Z 73,A -95.1344,B 24.9035,C -2.2679,E1 25.001,E2 -180.6009} C_DIS
LIN {X -0.3434,Y -68.3041,Z 73,A -95.1344,B 24.9035,C -2.2679,E1 25.001,E2 -180.6009} C_DIS
Enddeposition()
LIN {X 0.4529,Y -67.3416,Z 73,A -95.5497,B 24.9043,C -2.2585,E1 24.9998,E2 -180.1633} C_DIS
Startdeposition()
$VEL.CP = VEL_PRINT
LIN {X -3.3394,Y -67.2733,Z 73,A -99.9815,B 24.9067,C -2.2297,E1 24.9872,E2 -175.6622} C_DIS
LIN {X -7.6654,Y -66.9177,Z 73,A -102.0524,B 24.9035,C -2.2678,E1 24.9817,E2 -173.6808} C_DIS
LIN {X -10.7569,Y -66.4908,Z 73,A -105.1609,B 24.9044,C -2.2578,E1 24.973,E2 -170.5458} C_DIS
LIN {X -14.2657,Y -65.827,Z 73,A -108.4859,B 24.9048,C -2.2524,E1 24.9639,E2 -167.2042} C_DIS
LIN {X -16.9902,Y -65.1774,Z 73,A -110.9095,B 24.9048,C -2.2528,E1 24.9573,E2 -164.7781} C_DIS
LIN {X -20.9404,Y -64.0176,Z 73,A -114.1413,B 24.9041,C -2.2614,E1 24.9487,E2 -161.5613} C_DIS
LIN {X -24.3383,Y -62.8048,Z 73,A -117.3213,B 24.9041,C -2.2616,E1 24.9404,E2 -158.3752} C_DIS
LIN {X -29.1071,Y -60.7411,Z 73,A -121.613,B 24.9034,C -2.2693,E1 24.9295,E2 -154.0915} C_DIS
LIN {X -31.8184,Y -59.3667,Z 73,A -124.2049,B 24.9031,C -2.2724,E1 24.9231,E2 -151.4998} C_DIS
LIN {X -34.4736,Y -57.8648,Z 73,A -127.5679,B 24.9042,C -2.2593,E1 24.9149,E2 -148.0954} C_DIS
LIN {X -37.3285,Y -56.0658,Z 73,A -129.8379,B 24.9027,C -2.2768,E1 24.9097,E2 -145.8596} C_DIS
LIN {X -40.2051,Y -54.0403,Z 73,A -133.6284,B 24.9038,C -2.2647,E1 24.901,E2 -142.0269} C_DIS
LIN {X -43.1704,Y -51.7015,Z 73,A -135.9948,B 24.9017,C -2.2887,E1 24.896,E2 -139.7087} C_DIS
LIN {X -46.0659,Y -49.139,Z 73,A -139.4465,B 24.9015,C -2.2917,E1 24.8889,E2 -136.2502} C_DIS
LIN {X -48.9285,Y -46.2898,Z 73,A -142.7242,B 24.9006,C -2.3023,E1 24.8825,E2 -132.9838} C_DIS
LIN {X -50.8623,Y -44.1561,Z 73,A -145.0056,B 24.8998,C -2.3112,E1 24.8783,E2 -130.7136} C_DIS
LIN {X -52.0457,Y -42.7557,Z 73,A -146.6612,B 24.8996,C -2.3128,E1 24.8753,E2 -129.054} C_DIS
LIN {X -53.7031,Y -40.6539,Z 73,A -148.7593,B 24.8988,C -2.3219,E1 24.8718,E2 -126.9678} C_DIS
LIN {X -55.4369,Y -38.2558,Z 73,A -151.9625,B 24.8996,C -2.3138,E1 24.8666,E2 -123.7296} C_DIS
LIN {X -57.639,Y -34.8493,Z 73,A -154.9345,B 24.8979,C -2.3326,E1 24.8622,E2 -120.7871} C_DIS
LIN {X -58.7014,Y -33.0287,Z 73,A -157.2908,B 24.8985,C -2.3257,E1 24.8589,E2 -118.4022} C_DIS
LIN {X -61.2202,Y -28.0879,Z 73,A -161.5369,B 24.8965,C -2.3483,E1 24.8537,E2 -114.1871} C_DIS
LIN {X -62.6732,Y -24.6734,Z 73,A -165.0307,B 24.8963,C -2.3504,E1 24.85,E2 -110.6789} C_DIS
LIN {X -63.8177,Y -21.5407,Z 73,A -167.601,B 24.8951,C -2.3641,E1 24.8477,E2 -108.1267} C_DIS
LIN {X -64.6601,Y -18.8643,Z 73,A -170.1102,B 24.8947,C -2.3687,E1 24.8457,E2 -105.614} C_DIS
LIN {X -65.4567,Y -15.8784,Z 73,A -172.5269,B 24.8936,C -2.3809,E1 24.844,E2 -103.2124} C_DIS
LIN {X -65.9066,Y -13.8978,Z 73,A -174.6778,B 24.8939,C -2.3776,E1 24.8427,E2 -101.0409} C_DIS
LIN {X -66.5056,Y -10.6699,Z 73,A -177.503,B 24.8932,C -2.3856,E1 24.8414,E2 -98.218} C_DIS
LIN {X -66.9217,Y -7.6311,Z 73,A 179.5209,B 24.8932,C -2.3864,E1 24.8405,E2 -95.226} C_DIS
LIN {X -67.2668,Y -3.4558,Z 73,A 176.7563,B 24.8907,C -2.4136,E1 24.8399,E2 -92.5097} C_DIS
LIN {X -67.3522,Y -0.7005,Z 73,A 174.0614,B 24.8907,C -2.414,E1 24.8398,E2 -89.7994} C_DIS
LIN {X -67.3241,Y 2.0413,Z 73,A 171.3998,B 24.8906,C -2.4148,E1 24.84,E2 -87.1238} C_DIS
LIN {X -66.9415,Y 7.4588,Z 73,A 167.4598,B 24.888,C -2.443,E1 24.8409,E2 -83.2276} C_DIS
LIN {X -66.5758,Y 10.2159,Z 73,A 164.7839,B 24.8879,C -2.4443,E1 24.8419,E2 -80.5388} C_DIS
LIN {X -66.0916,Y 12.9873,Z 73,A 162.5035,B 24.887,C -2.4541,E1 24.8431,E2 -78.2682} C_DIS
LIN {X -65.4545,Y 15.8875,Z 73,A 160.0231,B 24.8862,C -2.4629,E1 24.8446,E2 -75.7943} C_DIS
LIN {X -64.6524,Y 18.8905,Z 73,A 156.6725,B 24.8867,C -2.4569,E1 24.8472,E2 -72.4101} C_DIS
LIN {X -63.2784,Y 23.077,Z 73,A 153.5756,B 24.8844,C -2.4814,E1 24.85,E2 -69.3542} C_DIS
LIN {X -62.2287,Y 25.777,Z 73,A 150.9229,B 24.8841,C -2.485,E1 24.8528,E2 -66.6952} C_DIS
LIN {X -61.0374,Y 28.4805,Z 73,A 147.9056,B 24.8843,C -2.4824,E1 24.8563,E2 -63.655} C_DIS
LIN {X -58.8994,Y 32.6742,Z 73,A 144.4321,B 24.8822,C -2.5046,E1 24.8608,E2 -60.2162} C_DIS
LIN {X -57.5207,Y 35.0438,Z 73,A 142.1402,B 24.8816,C -2.512,E1 24.8641,E2 -57.9303} C_DIS
LIN {X -55.8147,Y 37.7018,Z 73,A 139.197,B 24.8813,C -2.5142,E1 24.8686,E2 -54.9774} C_DIS
LIN {X -53.9672,Y 40.3023,Z 73,A 135.3266,B 24.8829,C -2.498,E1 24.8752,E2 -51.0498} C_DIS
LIN {X -51.0059,Y 43.9915,Z 73,A 131.9256,B 24.8807,C -2.5208,E1 24.8812,E2 -47.6877} C_DIS
LIN {X -47.4836,Y 47.7709,Z 73,A 127.2574,B 24.8802,C -2.5258,E1 24.8904,E2 -43.0114} C_DIS
LIN {X -44.7705,Y 50.3224,Z 73,A 125.116,B 24.8775,C -2.5542,E1 24.8947,E2 -40.9292} C_DIS
LIN {X -42.0851,Y 52.5897,Z 73,A 121.5939,B 24.878,C -2.5495,E1 24.9023,E2 -37.3825} C_DIS
LIN {X -39.4977,Y 54.5595,Z 73,A 118.3349,B 24.8784,C -2.5448,E1 24.9098,E2 -34.1009} C_DIS
LIN {X -36.5326,Y 56.5871,Z 73,A 116.4885,B 24.8754,C -2.5762,E1 24.9139,E2 -32.3232} C_DIS
LIN {X -32.877,Y 58.7861,Z 73,A 112.5532,B 24.8754,C -2.576,E1 24.9234,E2 -28.3757} C_DIS
LIN {X -30.4843,Y 60.062,Z 73,A 109.816,B 24.876,C -2.5705,E1 24.9302,E2 -25.6179} C_DIS
LIN {X -27.1378,Y 61.6465,Z 73,A 107.0461,B 24.8747,C -2.5834,E1 24.9372,E2 -22.8719} C_DIS
LIN {X -24.4057,Y 62.7784,Z 73,A 104.5233,B 24.8744,C -2.5867,E1 24.9437,E2 -20.3513} C_DIS
LIN {X -21.7468,Y 63.7482,Z 73,A 102.0508,B 24.8742,C -2.5882,E1 24.9502,E2 -17.8776} C_DIS
LIN {X -19.7403,Y 64.3978,Z 73,A 99.4703,B 24.8757,C -2.573,E1 24.9572,E2 -15.2565} C_DIS
LIN {X -16.3684,Y 65.3372,Z 73,A 97.5531,B 24.8731,C -2.5993,E1 24.9623,E2 -13.399} C_DIS
LIN {X -14.3244,Y 65.8142,Z 73,A 94.9831,B 24.8747,C -2.5834,E1 24.9694,E2 -10.788} C_DIS
LIN {X -9.2354,Y 66.7193,Z 73,A 91.1027,B 24.8733,C -2.5981,E1 24.98,E2 -6.9388} C_DIS
LIN {X -5.7759,Y 67.1081,Z 73,A 87.8266,B 24.8738,C -2.5924,E1 24.9891,E2 -3.6476} C_DIS
LIN {X -1.0504,Y 67.3471,Z 73,A 84.1153,B 24.873,C -2.6009,E1 24.9994,E2 0.0444} C_DIS
LIN {X 3.9422,Y 67.2397,Z 73,A 79.8396,B 24.873,C -2.6006,E1 25.0114,E2 4.3196} C_DIS
LIN {X 7.5692,Y 66.9287,Z 73,A 76.6188,B 24.8733,C -2.5974,E1 25.0203,E2 7.5461} C_DIS
LIN {X 11.0991,Y 66.4343,Z 73,A 73.5146,B 24.8736,C -2.5948,E1 25.0289,E2 10.6535} C_DIS
LIN {X 14.0556,Y 65.8729,Z 73,A 70.8994,B 24.8738,C -2.5924,E1 25.0361,E2 13.2712} C_DIS
LIN {X 17.8141,Y 64.9571,Z 73,A 67.8434,B 24.8735,C -2.596,E1 25.0443,E2 16.3141} C_DIS
LIN {X 21.311,Y 63.8952,Z 73,A 64.741,B 24.8737,C -2.5937,E1 25.0525,E2 19.416} C_DIS
LIN {X 25.7433,Y 62.2425,Z 73,A 60.7285,B 24.874,C -2.5902,E1 25.063,E2 23.4282} C_DIS
LIN {X 28.4513,Y 61.051,Z 73,A 58.1945,B 24.8744,C -2.5869,E1 25.0694,E2 25.9636} C_DIS
LIN {X 31.358,Y 59.6102,Z 73,A 55.7299,B 24.874,C -2.5907,E1 25.0755,E2 28.4125} C_DIS
LIN {X 35.4206,Y 57.2903,Z 73,A 51.6114,B 24.8749,C -2.5816,E1 25.0855,E2 32.5401} C_DIS
LIN {X 38.4339,Y 55.3131,Z 73,A 48.0136,B 24.8766,C -2.5635,E1 25.0939,E2 36.1687} C_DIS
LIN {X 41.7749,Y 52.8352,Z 73,A 45.1973,B 24.8755,C -2.5753,E1 25.1001,E2 38.9466} C_DIS
LIN {X 44.163,Y 50.8563,Z 73,A 42.1075,B 24.8771,C -2.5589,E1 25.1067,E2 42.0633} C_DIS
LIN {X 46.9973,Y 48.2502,Z 73,A 38.9335,B 24.8775,C -2.5549,E1 25.1131,E2 45.2339} C_DIS
LIN {X 48.7775,Y 46.4502,Z 73,A 37.0922,B 24.8771,C -2.5582,E1 25.1167,E2 47.0594} C_DIS
LIN {X 51.3856,Y 43.5459,Z 73,A 33.617,B 24.8782,C -2.5468,E1 25.1231,E2 50.5459} C_DIS
LIN {X 53.1612,Y 41.3605,Z 73,A 31.3734,B 24.8784,C -2.5451,E1 25.127,E2 52.7832} C_DIS
LIN {X 54.2247,Y 39.9553,Z 73,A 29.1532,B 24.8805,C -2.5229,E1 25.1308,E2 55.0451} C_DIS
LIN {X 56.3657,Y 36.8736,Z 73,A 26.2172,B 24.8807,C -2.5214,E1 25.1353,E2 57.97} C_DIS
LIN {X 58.2432,Y 33.8309,Z 73,A 23.6136,B 24.8803,C -2.5249,E1 25.139,E2 60.5522} C_DIS
LIN {X 60.161,Y 30.2907,Z 73,A 20.1013,B 24.8814,C -2.5133,E1 25.1436,E2 64.0733} C_DIS
LIN {X 61.403,Y 27.6835,Z 73,A 17.9209,B 24.8814,C -2.5137,E1 25.1461,E2 66.2409} C_DIS
LIN {X 62.4701,Y 25.1825,Z 73,A 15.3529,B 24.8826,C -2.5005,E1 25.1489,E2 68.8261} C_DIS
LIN {X 63.3008,Y 23.0156,Z 73,A 12.4016,B 24.8856,C -2.4691,E1 25.1518,E2 71.8349} C_DIS
LIN {X 64.573,Y 19.1581,Z 73,A 10.5939,B 24.8825,C -2.5023,E1 25.1532,E2 73.5539} C_DIS
LIN {X 65.6572,Y 15.0284,Z 73,A 6.4425,B 24.8848,C -2.4775,E1 25.1561,E2 77.7401} C_DIS
LIN {X 66.1481,Y 12.6938,Z 73,A 4.2017,B 24.8859,C -2.4656,E1 25.1573,E2 79.9958} C_DIS
LIN {X 66.7107,Y 9.2958,Z 73,A 1.5217,B 24.8861,C -2.4632,E1 25.1585,E2 82.6658} C_DIS
LIN {X 67.0888,Y 5.9863,Z 73,A -1.3779,B 24.8871,C -2.4526,E1 25.1593,E2 85.5733} C_DIS
LIN {X 67.2839,Y 3.1029,Z 73,A -4.6147,B 24.8897,C -2.4242,E1 25.1598,E2 88.8579} C_DIS
LIN {X 67.3536,Y -0.4328,Z 73,A -6.2984,B 24.8873,C -2.4499,E1 25.1598,E2 90.4708} C_DIS
LIN {X 67.2721,Y -3.3615,Z 73,A -9.2544,B 24.8892,C -2.4296,E1 25.1595,E2 93.4574} C_DIS
LIN {X 67.0512,Y -6.3942,Z 73,A -11.7932,B 24.8899,C -2.4226,E1 25.1589,E2 95.9975} C_DIS
LIN {X 66.7154,Y -9.263,Z 73,A -14.2669,B 24.8906,C -2.4144,E1 25.158,E2 98.476} C_DIS
LIN {X 66.2027,Y -12.4103,Z 73,A -17.886,B 24.8935,C -2.3818,E1 25.1562,E2 102.151} C_DIS
LIN {X 65.3971,Y -16.1229,Z 73,A -20.4471,B 24.8929,C -2.3894,E1 25.1545,E2 104.6793} C_DIS
LIN {X 64.2977,Y -20.063,Z 73,A -23.4534,B 24.8927,C -2.3912,E1 25.1522,E2 107.664} C_DIS
LIN {X 63.5406,Y -22.345,Z 73,A -25.752,B 24.8939,C -2.3782,E1 25.1501,E2 109.9805} C_DIS
LIN {X 62.4912,Y -25.1322,Z 73,A -28.2204,B 24.8944,C -2.3723,E1 25.1476,E2 112.4493} C_DIS
LIN {X 61.2726,Y -27.9726,Z 73,A -31.0742,B 24.8956,C -2.3584,E1 25.1443,E2 115.3202} C_DIS
LIN {X 59.0741,Y -32.3578,Z 73,A -34.5509,B 24.8951,C -2.3648,E1 25.1399,E2 118.7635} C_DIS
LIN {X 57.5401,Y -35.012,Z 73,A -37.8391,B 24.8973,C -2.3393,E1 25.1352,E2 122.0948} C_DIS
LIN {X 55.7151,Y -37.8488,Z 73,A -40.4803,B 24.8975,C -2.3374,E1 25.1311,E2 124.7275} C_DIS
LIN {X 53.8752,Y -40.4248,Z 73,A -43.0007,B 24.8977,C -2.3347,E1 25.127,E2 127.2422} C_DIS
LIN {X 52.1916,Y -42.5768,Z 73,A -45.4328,B 24.8985,C -2.3258,E1 25.1227,E2 129.684} C_DIS
LIN {X 50.139,Y -44.9754,Z 73,A -47.9253,B 24.8987,C -2.324,E1 25.1182,E2 132.1694} C_DIS
LIN {X 46.8002,Y -48.4402,Z 73,A -52.1081,B 24.8997,C -2.3118,E1 25.11,E2 136.3633} C_DIS
LIN {X 44.98,Y -50.1349,Z 73,A -54.2505,B 24.9002,C -2.3062,E1 25.1055,E2 138.5102} C_DIS
LIN {X 42.777,Y -52.0284,Z 73,A -56.755,B 24.9008,C -2.2999,E1 25.1001,E2 141.02} C_DIS
LIN {X 38.9053,Y -54.9832,Z 73,A -60.8376,B 24.9014,C -2.2929,E1 25.091,E2 145.1046} C_DIS
LIN {X 36.0098,Y -56.9223,Z 73,A -64.0781,B 24.9025,C -2.2802,E1 25.0834,E2 148.3646} C_DIS
LIN {X 32.5622,Y -58.9619,Z 73,A -67.2779,B 24.9025,C -2.2794,E1 25.0756,E2 151.5567} C_DIS
LIN {X 29.6179,Y -60.4946,Z 73,A -69.6171,B 24.9019,C -2.287,E1 25.0699,E2 153.8714} C_DIS
LIN {X 27.4782,Y -61.4953,Z 73,A -72.0016,B 24.9029,C -2.2745,E1 25.0637,E2 156.2795} C_DIS
LIN {X 24.9796,Y -62.5525,Z 73,A -74.1563,B 24.9029,C -2.2751,E1 25.0582,E2 158.4279} C_DIS
LIN {X 21.7999,Y -63.7303,Z 73,A -77.1752,B 24.9035,C -2.268,E1 25.0502,E2 161.4574} C_DIS
LIN {X 18.619,Y -64.731,Z 73,A -79.8863,B 24.9035,C -2.2679,E1 25.043,E2 164.164} C_DIS
LIN {X 14.335,Y -65.8119,Z 73,A -83.6887,B 24.9039,C -2.2632,E1 25.0327,E2 167.9721} C_DIS
LIN {X 11.5338,Y -66.3603,Z 73,A -86.5112,B 24.9049,C -2.2517,E1 25.0248,E2 170.8188} C_DIS
LIN {X 7.8046,Y -66.9013,Z 73,A -89.9924,B 24.9056,C -2.2431,E1 25.0152,E2 174.3177} C_DIS
LIN {X 3.0999,Y -67.284,Z 73,A -93.2898,B 24.9043,C -2.2585,E1 25.0061,E2 177.5771} C_DIS
LIN {X 1.2058,Y -67.3443,Z 73,A -95.5141,B 24.9056,C -2.2435,E1 24.9998,E2 179.8367} C_DIS
LIN {X 1.2058,Y -67.3443,Z 73,A -95.5141,B 24.9056,C -2.2435,E1 24.9998,E2 179.8367} C_DIS
Enddeposition()
LIN {X 0.4624,Y -66.4029,Z 73,A -95.9452,B 24.9038,C -2.2649,E1 24.9987,E2 180.2169} C_DIS
Startdeposition()
$VEL.CP = VEL_PRINT
LIN {X 2.8181,Y -66.3453,Z 73,A -92.3941,B 24.9006,C -2.3014,E1 25.0089,E2 176.5796} C_DIS
LIN {X 8.0737,Y -65.9127,Z 73,A -88.1588,B 24.9011,C -2.2961,E1 25.0206,E2 172.3594} C_DIS
LIN {X 11.9532,Y -65.3204,Z 73,A -84.5765,B 24.9005,C -2.3033,E1 25.0305,E2 168.7635} C_DIS
LIN {X 15.6468,Y -64.5354,Z 73,A -81.112,B 24.8998,C -2.3114,E1 25.04,E2 165.2846} C_DIS
LIN {X 19.0331,Y -63.6192,Z 73,A -78.1971,B 24.8998,C -2.3119,E1 25.0478,E2 162.3733} C_DIS
LIN {X 21.6103,Y -62.7917,Z 73,A -75.157,B 24.8979,C -2.3325,E1 25.0559,E2 159.2904} C_DIS
LIN {X 25.7356,Y -61.2154,Z 73,A -71.8654,B 24.8986,C -2.3247,E1 25.0644,E2 156.0248} C_DIS
LIN {X 28.8424,Y -59.8145,Z 73,A -69.3706,B 24.8992,C -2.3179,E1 25.0707,E2 153.5523} C_DIS
LIN {X 31.6638,Y -58.3699,Z 73,A -66.1442,B 24.8977,C -2.335,E1 25.0787,E2 150.2945} C_DIS
LIN {X 36.6007,Y -55.4079,Z 73,A -62.0994,B 24.899,C -2.3206,E1 25.0883,E2 146.2966} C_DIS
LIN {X 39.5411,Y -53.3489,Z 73,A -58.3263,B 24.8969,C -2.3442,E1 25.0969,E2 142.4808} C_DIS
LIN {X 42.1102,Y -51.347,Z 73,A -55.6402,B 24.8966,C -2.347,E1 25.1028,E2 139.7981} C_DIS
LIN {X 44.0311,Y -49.7091,Z 73,A -53.5272,B 24.8964,C -2.3502,E1 25.1072,E2 137.6857} C_DIS
LIN {X 45.8614,Y -48.0257,Z 73,A -50.7524,B 24.8944,C -2.3717,E1 25.1129,E2 134.8715} C_DIS
LIN {X 48.6527,Y -45.1963,Z 73,A -47.9166,B 24.8951,C -2.3645,E1 25.1183,E2 132.0651} C_DIS
LIN {X 50.43,Y -43.2029,Z 73,A -45.5147,B 24.8943,C -2.3729,E1 25.1228,E2 129.6541} C_DIS
LIN {X 52.064,Y -41.2187,Z 73,A -43.5536,B 24.8944,C -2.3719,E1 25.1262,E2 127.7045} C_DIS
LIN {X 53.5861,Y -39.2196,Z 73,A -40.3015,B 24.8913,C -2.4066,E1 25.1317,E2 124.3861} C_DIS
LIN {X 55.7089,Y -36.1423,Z 73,A -38.1233,B 24.893,C -2.3875,E1 25.1349,E2 122.2639} C_DIS
LIN {X 58.1019,Y -32.1539,Z 73,A -33.8806,B 24.8915,C -2.405,E1 25.141,E2 118.0016} C_DIS
LIN {X 59.6297,Y -29.2237,Z 73,A -31.1743,B 24.8911,C -2.4095,E1 25.1443,E2 115.2992} C_DIS
LIN {X 61.0772,Y -26.0634,Z 73,A -28.4134,B 24.8908,C -2.4121,E1 25.1475,E2 112.5471} C_DIS
LIN {X 61.9709,Y -23.8617,Z 73,A -25.6759,B 24.8886,C -2.4367,E1 25.1503,E2 109.7666} C_DIS
LIN {X 63.3439,Y -19.9315,Z 73,A -22.1148,B 24.8876,C -2.4469,E1 25.1534,E2 106.2015} C_DIS
LIN {X 64.4743,Y -15.8978,Z 73,A -18.4555,B 24.8865,C -2.4594,E1 25.1559,E2 102.5338} C_DIS
LIN {X 65.3505,Y -11.7878,Z 73,A -14.9928,B 24.8858,C -2.4664,E1 25.1578,E2 99.0748} C_DIS
LIN {X 65.9518,Y -7.7465,Z 73,A -11.8689,B 24.8858,C -2.4667,E1 25.1589,E2 95.9685} C_DIS
LIN {X 66.2346,Y -4.7644,Z 73,A -8.3601,B 24.8827,C -2.5,E1 25.1596,E2 92.4021} C_DIS
LIN {X 66.4004,Y -0.8665,Z 73,A -5.3752,B 24.8827,C -2.5002,E1 25.1598,E2 89.4343} C_DIS
LIN {X 66.2191,Y 4.9766,Z 73,A -0.4643,B 24.8815,C -2.5125,E1 25.159,E2 84.5236} C_DIS
LIN {X 65.6929,Y 9.7071,Z 73,A 2.9662,B 24.882,C -2.5071,E1 25.1579,E2 81.1261} C_DIS
LIN {X 65.3304,Y 11.8995,Z 73,A 5.4011,B 24.8801,C -2.5269,E1 25.1566,E2 78.6587} C_DIS
LIN {X 64.2265,Y 16.8696,Z 73,A 9.6075,B 24.8793,C -2.5352,E1 25.1539,E2 74.457} C_DIS
LIN {X 63.2279,Y 20.2914,Z 73,A 12.6212,B 24.8786,C -2.5427,E1 25.1514,E2 71.4428} C_DIS
LIN {X 62.1249,Y 23.4551,Z 73,A 15.9543,B 24.8767,C -2.5628,E1 25.1482,E2 68.0807} C_DIS
LIN {X 60.4842,Y 27.4102,Z 73,A 18.7253,B 24.8781,C -2.5487,E1 25.1451,E2 65.3581} C_DIS
LIN {X 59.448,Y 29.5903,Z 73,A 21.827,B 24.8749,C -2.5814,E1 25.1412,E2 62.1958} C_DIS
LIN {X 57.8261,Y 32.6478,Z 73,A 23.6775,B 24.877,C -2.5594,E1 25.1388,E2 60.4069} C_DIS
LIN {X 55.6813,Y 36.1853,Z 73,A 27.5437,B 24.8754,C -2.5763,E1 25.1331,E2 56.5203} C_DIS
LIN {X 54.19,Y 38.3815,Z 73,A 29.6964,B 24.8752,C -2.5785,E1 25.1297,E2 54.3732} C_DIS
LIN {X 52.561,Y 40.583,Z 73,A 32.4588,B 24.8736,C -2.5945,E1 25.125,E2 51.5859} C_DIS
LIN {X 48.7835,Y 45.0539,Z 73,A 37.2043,B 24.8733,C -2.598,E1 25.1163,E2 46.8536} C_DIS
LIN {X 47.0551,Y 46.8565,Z 73,A 39.3658,B 24.8728,C -2.6027,E1 25.1121,E2 44.6901} C_DIS
LIN {X 44.5527,Y 49.2417,Z 73,A 42.5375,B 24.8718,C -2.6135,E1 25.1055,E2 41.5058} C_DIS
LIN {X 41.369,Y 51.9451,Z 73,A 45.8215,B 24.8718,C -2.6121,E1 25.0985,E2 38.2377} C_DIS
LIN {X 38.2751,Y 54.2659,Z 73,A 49.6567,B 24.8701,C -2.6303,E1 25.0898,E2 34.3729} C_DIS
LIN {X 34.7234,Y 56.6039,Z 73,A 53.3639,B 24.8694,C -2.6369,E1 25.081,E2 30.6621} C_DIS
LIN {X 29.3197,Y 59.5822,Z 73,A 58.0415,B 24.8703,C -2.6278,E1 25.0696,E2 26.0193} C_DIS
LIN {X 26.9154,Y 60.7072,Z 73,A 61.808,B 24.8665,C -2.6668,E1 25.0598,E2 22.1694} C_DIS
LIN {X 22.5519,Y 62.4588,Z 73,A 64.707,B 24.8689,C -2.642,E1 25.0523,E2 19.3354} C_DIS
LIN {X 18.774,Y 63.6959,Z 73,A 67.8713,B 24.8693,C -2.6382,E1 25.0439,E2 16.186} C_DIS
LIN {X 16.0254,Y 64.4425,Z 73,A 70.5416,B 24.8687,C -2.6448,E1 25.0367,E2 13.5041} C_DIS
LIN {X 13.5804,Y 65.0021,Z 73,A 72.5039,B 24.869,C -2.641,E1 25.0314,E2 11.5534} C_DIS
LIN {X 10.877,Y 65.5083,Z 73,A 74.8653,B 24.869,C -2.6416,E1 25.0249,E2 9.1932} C_DIS
LIN {X 8.1835,Y 65.8999,Z 73,A 77.3498,B 24.8686,C -2.6453,E1 25.018,E2 6.7018} C_DIS
LIN {X 4.9398,Y 66.222,Z 73,A 79.925,B 24.8691,C -2.64,E1 25.0109,E2 4.1407} C_DIS
LIN {X 3.0183,Y 66.3367,Z 73,A 81.9117,B 24.8684,C -2.6475,E1 25.0053,E2 2.1368} C_DIS
LIN {X -0.7772,Y 66.4011,Z 73,A 84.7348,B 24.8695,C -2.6365,E1 24.9975,E2 -0.6598} C_DIS
LIN {X -4.1977,Y 66.2729,Z 73,A 88.5541,B 24.8676,C -2.6553,E1 24.9867,E2 -4.5251} C_DIS
LIN {X -7.7944,Y 65.9461,Z 73,A 91.3278,B 24.8686,C -2.6458,E1 24.979,E2 -7.2778} C_DIS
LIN {X -11.439,Y 65.4133,Z 73,A 94.1428,B 24.8696,C -2.6354,E1 24.9713,E2 -10.0705} C_DIS
LIN {X -13.4778,Y 65.0231,Z 73,A 96.3791,B 24.8687,C -2.644,E1 24.9652,E2 -12.3297} C_DIS
LIN {X -16.1387,Y 64.4154,Z 73,A 99.4518,B 24.8673,C -2.6579,E1 24.9568,E2 -15.44} C_DIS
LIN {X -19.8702,Y 63.363,Z 73,A 101.8381,B 24.8699,C -2.6327,E1 24.9505,E2 -17.7705} C_DIS
LIN {X -22.2933,Y 62.552,Z 73,A 104.0424,B 24.8701,C -2.63,E1 24.9447,E2 -19.9725} C_DIS
LIN {X -25.0577,Y 61.496,Z 73,A 106.5932,B 24.8705,C -2.6265,E1 24.9381,E2 -22.5206} C_DIS
LIN {X -28.39,Y 60.0308,Z 73,A 109.7742,B 24.8708,C -2.6227,E1 24.93,E2 -25.7003} C_DIS
LIN {X -31.6094,Y 58.3994,Z 73,A 112.7005,B 24.8717,C -2.6136,E1 24.9228,E2 -28.6128} C_DIS
LIN {X -35.1752,Y 56.3236,Z 73,A 116.3246,B 24.8722,C -2.6086,E1 24.9141,E2 -32.2361} C_DIS
LIN {X -38.1743,Y 54.336,Z 73,A 119.4638,B 24.8728,C -2.6033,E1 24.9068,E2 -35.3732} C_DIS
LIN {X -39.9813,Y 53.0203,Z 73,A 121.8054,B 24.8723,C -2.6081,E1 24.9016,E2 -37.7347} C_DIS
LIN {X -43.2118,Y 50.4224,Z 73,A 125.335,B 24.8731,C -2.5994,E1 24.894,E2 -41.2568} C_DIS
LIN {X -46.5151,Y 47.3923,Z 73,A 128.8843,B 24.8747,C -2.5837,E1 24.8868,E2 -44.7834} C_DIS
LIN {X -49.9319,Y 43.7774,Z 73,A 132.9929,B 24.8761,C -2.5694,E1 24.8791,E2 -48.8757} C_DIS
LIN {X -51.7277,Y 41.6406,Z 73,A 135.9201,B 24.8756,C -2.5739,E1 24.8738,E2 -51.8274} C_DIS
LIN {X -53.6406,Y 39.1451,Z 73,A 138.4643,B 24.8767,C -2.5632,E1 24.8696,E2 -54.3583} C_DIS
LIN {X -55.7289,Y 36.1112,Z 73,A 141.8785,B 24.877,C -2.5594,E1 24.8643,E2 -57.7804} C_DIS
LIN {X -57.3204,Y 33.5277,Z 73,A 144.3107,B 24.8781,C -2.5482,E1 24.8608,E2 -60.1984} C_DIS
LIN {X -59.1325,Y 30.2158,Z 73,A 147.7867,B 24.8786,C -2.5433,E1 24.8563,E2 -63.6811} C_DIS
LIN {X -61.1093,Y 25.9873,Z 73,A 151.5811,B 24.8802,C -2.5266,E1 24.8519,E2 -67.4564} C_DIS
LIN {X -62.2054,Y 23.2425,Z 73,A 154.5644,B 24.8801,C -2.5277,E1 24.8489,E2 -70.4591} C_DIS
LIN {X -63.5991,Y 19.1011,Z 73,A 158.1847,B 24.8815,C -2.513,E1 24.8459,E2 -74.0651} C_DIS
LIN {X -64.5073,Y 15.7623,Z 73,A 161.4205,B 24.8819,C -2.5088,E1 24.8437,E2 -77.3098} C_DIS
LIN {X -65.3633,Y 11.7165,Z 73,A 164.9161,B 24.883,C -2.4961,E1 24.8418,E2 -80.7957} C_DIS
LIN {X -65.9079,Y 8.1174,Z 73,A 167.7325,B 24.8846,C -2.4796,E1 24.8408,E2 -83.5895} C_DIS
LIN {X -66.2563,Y 4.4436,Z 73,A 171.2481,B 24.8849,C -2.4763,E1 24.84,E2 -87.1182} C_DIS
LIN {X -66.3914,Y 1.3561,Z 73,A 173.4413,B 24.8866,C -2.4583,E1 24.8398,E2 -89.2815} C_DIS
LIN {X -66.3888,Y -1.4977,Z 73,A 176.1861,B 24.8868,C -2.4562,E1 24.8398,E2 -92.0379} C_DIS
LIN {X -66.234,Y -4.7699,Z 73,A 179.4373,B 24.8868,C -2.4559,E1 24.8405,E2 -95.308} C_DIS
LIN {X -65.8306,Y -8.7184,Z 73,A -177.6562,B 24.8887,C -2.4347,E1 24.8414,E2 -98.1813} C_DIS
LIN {X -65.4985,Y -10.9354,Z 73,A -174.8989,B 24.8878,C -2.4456,E1 24.8427,E2 -100.9809} C_DIS
LIN {X -64.8776,Y -14.1614,Z 73,A -172.9815,B 24.8903,C -2.4182,E1 24.8438,E2 -102.844} C_DIS
LIN {X -64.3652,Y -16.334,Z 73,A -170.8517,B 24.8904,C -2.4165,E1 24.8452,E2 -104.9823} C_DIS
LIN {X -63.5316,Y -19.3264,Z 73,A -167.8071,B 24.8904,C -2.416,E1 24.8476,E2 -108.0434} C_DIS
LIN {X -62.5747,Y -22.2288,Z 73,A -165.2288,B 24.8913,C -2.4071,E1 24.85,E2 -110.615} C_DIS
LIN {X -61.0643,Y -26.0933,Z 73,A -162.1796,B 24.8932,C -2.3859,E1 24.8531,E2 -113.6308} C_DIS
LIN {X -60.3921,Y -27.6146,Z 73,A -159.9652,B 24.8921,C -2.3981,E1 24.8557,E2 -115.8862} C_DIS
LIN {X -57.7967,Y -32.7006,Z 73,A -155.4273,B 24.894,C -2.3767,E1 24.8617,E2 -120.3971} C_DIS
LIN {X -55.7564,Y -36.0683,Z 73,A -151.4233,B 24.8936,C -2.3808,E1 24.8677,E2 -124.4312} C_DIS
LIN {X -52.8648,Y -40.1884,Z 73,A -147.2771,B 24.895,C -2.366,E1 24.8745,E2 -128.5624} C_DIS
LIN {X -50.9825,Y -42.5493,Z 73,A -145.0624,B 24.8962,C -2.3517,E1 24.8784,E2 -130.7531} C_DIS
LIN {X -49.1432,Y -44.6619,Z 73,A -142.7031,B 24.8968,C -2.3451,E1 24.8827,E2 -133.1073} C_DIS
LIN {X -46.2381,Y -47.6623,Z 73,A -138.832,B 24.897,C -2.3434,E1 24.8904,E2 -136.9906} C_DIS
LIN {X -42.995,Y -50.6071,Z 73,A -135.2398,B 24.898,C -2.332,E1 24.8979,E2 -140.57} C_DIS
LIN {X -39.6797,Y -53.2469,Z 73,A -131.8302,B 24.899,C -2.3201,E1 24.9053,E2 -143.9638} C_DIS
LIN {X -37.1071,Y -55.0702,Z 73,A -129.2446,B 24.8996,C -2.3128,E1 24.9112,E2 -146.5406} C_DIS
LIN {X -35.3328,Y -56.2252,Z 73,A -127.0803,B 24.8992,C -2.3174,E1 24.9164,E2 -148.7229} C_DIS
LIN {X -32.7818,Y -57.7494,Z 73,A -124.2124,B 24.899,C -2.3206,E1 24.9233,E2 -151.607} C_DIS
LIN {X -30.5571,Y -58.958,Z 73,A -121.6657,B 24.8985,C -2.326,E1 24.9297,E2 -154.1735} C_DIS
LIN {X -25.6924,Y -61.2336,Z 73,A -118.2223,B 24.9013,C -2.294,E1 24.9383,E2 -157.5493} C_DIS
LIN {X -23.5807,Y -62.0774,Z 73,A -115.4869,B 24.8999,C -2.3097,E1 24.9455,E2 -160.3277} C_DIS
LIN {X -20.6336,Y -63.1184,Z 73,A -112.8462,B 24.9002,C -2.3062,E1 24.9525,E2 -162.9652} C_DIS
LIN {X -17.2141,Y -64.1352,Z 73,A -109.791,B 24.9004,C -2.3037,E1 24.9607,E2 -166.0193} C_DIS
LIN {X -13.8637,Y -64.9416,Z 73,A -106.9049,B 24.9007,C -2.3002,E1 24.9685,E2 -168.901} C_DIS
LIN {X -10.8103,Y -65.5195,Z 73,A -103.9772,B 24.9003,C -2.3051,E1 24.9766,E2 -171.8432} C_DIS
LIN {X -7.8037,Y -65.9451,Z 73,A -101.7954,B 24.9012,C -2.2944,E1 24.9826,E2 -174.001} C_DIS
LIN {X -3.1654,Y -66.3293,Z 73,A -97.6378,B 24.901,C -2.2977,E1 24.9942,E2 -178.1682} C_DIS
LIN {X 0.4624,Y -66.4029,Z 73,A -95.9438,B 24.9038,C -2.2643,E1 24.9987,E2 -179.7831} C_DIS
Enddeposition()
LIN {X 0.4624,Y -66.4029,Z 73,A -95.9438,B 24.9038,C -2.2643,E1 24.9987,E2 -179.7831} C_DIS
Startdeposition()
$VEL.CP = VEL_PRINT
LIN {X -1.4841,Y -65.439,Z 73,A -97.0757,B 24.9013,C -2.2939,E1 24.9957,E2 -178.7215} C_DIS
LIN {X -5.9645,Y -65.1829,Z 73,A -101.3258,B 24.9019,C -2.2865,E1 24.9839,E2 -174.4522} C_DIS
LIN {X -8.0426,Y -64.9603,Z 73,A -103.486,B 24.9025,C -2.2793,E1 24.9778,E2 -172.2733} C_DIS
LIN {X -11.5452,Y -64.429,Z 73,A -106.0706,B 24.9015,C -2.2918,E1 24.9708,E2 -169.7162} C_DIS
LIN {X -14.9013,Y -63.7367,Z 73,A -109.1388,B 24.9015,C -2.2916,E1 24.9624,E2 -166.6437} C_DIS
LIN {X -17.4387,Y -63.0899,Z 73,A -111.5517,B 24.9015,C -2.2903,E1 24.9558,E2 -164.2239} C_DIS
LIN {X -20.3269,Y -62.2193,Z 73,A -114.6373,B 24.9023,C -2.2825,E1 24.9476,E2 -161.1143} C_DIS
LIN {X -25.159,Y -60.4276,Z 73,A -118.3123,B 24.9003,C -2.3049,E1 24.9381,E2 -157.485} C_DIS
LIN {X -29.1082,Y -58.6268,Z 73,A -122.4343,B 24.9006,C -2.3021,E1 24.9276,E2 -153.3461} C_DIS
LIN {X -30.7391,Y -57.7888,Z 73,A -124.3211,B 24.9009,C -2.2981,E1 24.9229,E2 -151.4446} C_DIS
LIN {X -33.9372,Y -55.9701,Z 73,A -127.7759,B 24.9009,C -2.2977,E1 24.9146,E2 -147.9783} C_DIS
LIN {X -36.416,Y -54.391,Z 73,A -130.4949,B 24.9009,C -2.2987,E1 24.9083,E2 -145.2526} C_DIS
LIN {X -39.1543,Y -52.4535,Z 73,A -132.9955,B 24.8996,C -2.3127,E1 24.9027,E2 -142.7766} C_DIS
LIN {X -42.2303,Y -50.0107,Z 73,A -137.2662,B 24.9006,C -2.3019,E1 24.8934,E2 -138.4638} C_DIS
LIN {X -45.0063,Y -47.5276,Z 73,A -138.9418,B 24.8972,C -2.3411,E1 24.8902,E2 -136.8749} C_DIS
LIN {X -47.5757,Y -44.9551,Z 73,A -142.7855,B 24.8978,C -2.334,E1 24.8826,E2 -132.9979} C_DIS
LIN {X -49.0485,Y -43.3449,Z 73,A -144.7545,B 24.8975,C -2.337,E1 24.8789,E2 -131.0273} C_DIS
LIN {X -51.9563,Y -39.8116,Z 73,A -148.4144,B 24.8961,C -2.3533,E1 24.8725,E2 -127.3893} C_DIS
LIN {X -53.8636,Y -37.1905,Z 73,A -151.7466,B 24.8964,C -2.3503,E1 24.867,E2 -124.0335} C_DIS
LIN {X -56.3135,Y -33.3643,Z 73,A -155.6146,B 24.8953,C -2.3627,E1 24.8613,E2 -120.1754} C_DIS
LIN {X -58.2299,Y -29.8944,Z 73,A -159.3837,B 24.895,C -2.3661,E1 24.8564,E2 -116.3944} C_DIS
LIN {X -59.8602,Y -26.4816,Z 73,A -162.8541,B 24.8944,C -2.3721,E1 24.8523,E2 -112.9195} C_DIS
LIN {X -61.7423,Y -21.7321,Z 73,A -166.3603,B 24.8915,C -2.404,E1 24.8489,E2 -109.4698} C_DIS
LIN {X -62.7646,Y -18.5741,Z 73,A -169.7439,B 24.8916,C -2.4032,E1 24.846,E2 -106.0647} C_DIS
LIN {X -63.4268,Y -16.1694,Z 73,A -171.963,B 24.8911,C -2.409,E1 24.8444,E2 -103.8466} C_DIS
LIN {X -64.2838,Y -12.3279,Z 73,A -175.867,B 24.8909,C -2.4106,E1 24.8422,E2 -99.9235} C_DIS
LIN {X -64.839,Y -8.9638,Z 73,A -178.6322,B 24.8897,C -2.4241,E1 24.841,E2 -97.174} C_DIS
LIN {X -65.1792,Y -6.0053,Z 73,A 179.0682,B 24.8884,C -2.4382,E1 24.8404,E2 -94.8943} C_DIS
LIN {X -65.3909,Y -2.9039,Z 73,A 175.6722,B 24.8888,C -2.4337,E1 24.8398,E2 -91.4672} C_DIS
LIN {X -65.4119,Y 2.4047,Z 73,A 171.2879,B 24.887,C -2.4534,E1 24.84,E2 -87.1036} C_DIS
LIN {X -65.179,Y 6.0073,Z 73,A 168.4289,B 24.8856,C -2.4693,E1 24.8406,E2 -84.2653} C_DIS
LIN {X -64.9254,Y 8.3116,Z 73,A 165.8813,B 24.8859,C -2.4657,E1 24.8414,E2 -81.6939} C_DIS
LIN {X -64.4206,Y 11.5919,Z 73,A 163.5903,B 24.8839,C -2.4867,E1 24.8425,E2 -79.4395} C_DIS
LIN {X -63.5601,Y 15.6371,Z 73,A 159.7734,B 24.8832,C -2.4942,E1 24.8448,E2 -75.6181} C_DIS
LIN {X -62.5413,Y 19.3126,Z 73,A 156.3809,B 24.8824,C -2.5035,E1 24.8474,E2 -72.2281} C_DIS
LIN {X -60.9502,Y 23.8634,Z 73,A 152.2583,B 24.881,C -2.5182,E1 24.8513,E2 -68.1174} C_DIS
LIN {X -59.0749,Y 28.1883,Z 73,A 147.9342,B 24.8802,C -2.5266,E1 24.8562,E2 -63.7894} C_DIS
LIN {X -56.9568,Y 32.2563,Z 73,A 143.8132,B 24.8793,C -2.5361,E1 24.8616,E2 -59.6693} C_DIS
LIN {X -54.6416,Y 36.0372,Z 73,A 140.3213,B 24.8775,C -2.5546,E1 24.8667,E2 -56.2038} C_DIS
LIN {X -52.9792,Y 38.4405,Z 73,A 137.5476,B 24.8772,C -2.5572,E1 24.8711,E2 -53.4226} C_DIS
LIN {X -51.8963,Y 39.8895,Z 73,A 135.6674,B 24.8774,C -2.5555,E1 24.8743,E2 -51.5294} C_DIS
LIN {X -49.7753,Y 42.5066,Z 73,A 132.8152,B 24.8765,C -2.5649,E1 24.8794,E2 -48.6866} C_DIS
LIN {X -47.2243,Y 45.3241,Z 73,A 129.5378,B 24.8756,C -2.5741,E1 24.8856,E2 -45.4167} C_DIS
LIN {X -45.3686,Y 47.1814,Z 73,A 126.9069,B 24.8757,C -2.5728,E1 24.8909,E2 -42.7717} C_DIS
LIN {X -42.5382,Y 49.7484,Z 73,A 123.6764,B 24.8748,C -2.5826,E1 24.8976,E2 -39.5518} C_DIS
LIN {X -39.7984,Y 51.9664,Z 73,A 120.5981,B 24.8741,C -2.5893,E1 24.9043,E2 -36.4781} C_DIS
LIN {X -36.8319,Y 54.1094,Z 73,A 117.6333,B 24.873,C -2.6005,E1 24.9111,E2 -33.5299} C_DIS
LIN {X -34.3993,Y 55.6879,Z 73,A 114.5231,B 24.8737,C -2.5935,E1 24.9185,E2 -30.393} C_DIS
LIN {X -31.5554,Y 57.348,Z 73,A 111.9513,B 24.8726,C -2.6048,E1 24.9247,E2 -27.8407} C_DIS
LIN {X -29.1956,Y 58.5835,Z 73,A 109.3498,B 24.8728,C -2.603,E1 24.9312,E2 -25.2279} C_DIS
LIN {X -24.6942,Y 60.6183,Z 73,A 105.2886,B 24.8716,C -2.6147,E1 24.9415,E2 -21.185} C_DIS
LIN {X -20.0105,Y 62.3216,Z 73,A 101.1138,B 24.8707,C -2.6241,E1 24.9525,E2 -17.0243} C_DIS
LIN {X -15.9089,Y 63.4937,Z 73,A 97.4841,B 24.8701,C -2.6302,E1 24.9622,E2 -13.4034} C_DIS
LIN {X -12.625,Y 64.2263,Z 73,A 94.3258,B 24.8703,C -2.6281,E1 24.9709,E2 -10.2363} C_DIS
LIN {X -8.9239,Y 64.8445,Z 73,A 91.0103,B 24.8702,C -2.6296,E1 24.98,E2 -6.9216} C_DIS
LIN {X -6.3027,Y 65.1517,Z 73,A 88.3126,B 24.8709,C -2.6223,E1 24.9876,E2 -4.2049} C_DIS
LIN {X -1.7364,Y 65.4328,Z 73,A 84.9163,B 24.8694,C -2.6372,E1 24.9969,E2 -0.8431} C_DIS
LIN {X -0.0345,Y 65.4563,Z 73,A 82.8559,B 24.8706,C -2.6248,E1 25.0028,E2 1.2468} C_DIS
LIN {X 3.6482,Y 65.3535,Z 73,A 79.9099,B 24.87,C -2.6312,E1 25.011,E2 4.1766} C_DIS
LIN {X 6.5213,Y 65.1302,Z 73,A 77.3924,B 24.87,C -2.6312,E1 25.018,E2 6.6929} C_DIS
LIN {X 9.7898,Y 64.7193,Z 73,A 74.4111,B 24.8703,C -2.6282,E1 25.0262,E2 9.6786} C_DIS
LIN {X 13.4312,Y 64.063,Z 73,A 71.4294,B 24.8698,C -2.6328,E1 25.0344,E2 12.6458} C_DIS
LIN {X 15.9315,Y 63.4875,Z 73,A 69.0742,B 24.8702,C -2.6291,E1 25.0408,E2 15.0067} C_DIS
LIN {X 19.7821,Y 62.3955,Z 73,A 65.0327,B 24.8717,C -2.6141,E1 25.0516,E2 19.0766} C_DIS
LIN {X 24.6236,Y 60.6471,Z 73,A 60.6683,B 24.8717,C -2.6132,E1 25.063,E2 23.4337} C_DIS
LIN {X 27.6311,Y 59.3373,Z 73,A 58.2523,B 24.871,C -2.6207,E1 25.0691,E2 25.8259} C_DIS
LIN {X 30.8023,Y 57.7557,Z 73,A 54.7438,B 24.8724,C -2.607,E1 25.0779,E2 29.3569} C_DIS
LIN {X 34.0254,Y 55.9165,Z 73,A 51.5234,B 24.8728,C -2.603,E1 25.0856,E2 32.577} C_DIS
LIN {X 39.0078,Y 52.5622,Z 73,A 46.6467,B 24.8728,C -2.6037,E1 25.0967,E2 37.4355} C_DIS
LIN {X 41.7044,Y 50.4496,Z 73,A 43.7515,B 24.873,C -2.6007,E1 25.103,E2 40.3268} C_DIS
LIN {X 43.4383,Y 48.9651,Z 73,A 41.1336,B 24.8749,C -2.5817,E1 25.1086,E2 42.9795} C_DIS
LIN {X 46.8026,Y 45.7605,Z 73,A 37.3731,B 24.8749,C -2.5808,E1 25.116,E2 46.7263} C_DIS
LIN {X 49.4901,Y 42.8385,Z 73,A 34.1111,B 24.8752,C -2.5783,E1 25.1221,E2 49.9795} C_DIS
LIN {X 51.2047,Y 40.7734,Z 73,A 31.2712,B 24.8769,C -2.5606,E1 25.1271,E2 52.8481} C_DIS
LIN {X 53.9175,Y 37.113,Z 73,A 27.6111,B 24.8771,C -2.559,E1 25.133,E2 56.4941} C_DIS
LIN {X 56.6311,Y 32.8233,Z 73,A 23.4333,B 24.8775,C -2.5543,E1 25.1391,E2 60.662} C_DIS
LIN {X 58.0642,Y 30.2154,Z 73,A 20.65,B 24.8786,C -2.5427,E1 25.1428,E2 63.458} C_DIS
LIN {X 59.3815,Y 27.536,Z 73,A 17.818,B 24.8799,C -2.5299,E1 25.1462,E2 66.305} C_DIS
LIN {X 61.1852,Y 23.2545,Z 73,A 14.021,B 24.8803,C -2.5252,E1 25.1502,E2 70.0922} C_DIS
LIN {X 62.3552,Y 19.9043,Z 73,A 11.1447,B 24.8806,C -2.522,E1 25.1527,E2 72.9598} C_DIS
LIN {X 63.2312,Y 16.9183,Z 73,A 7.9962,B 24.8824,C -2.5029,E1 25.1551,E2 76.1353} C_DIS
LIN {X 64.0661,Y 13.416,Z 73,A 4.8926,B 24.8832,C -2.4945,E1 25.157,E2 79.2407} C_DIS
LIN {X 64.7504,Y 9.5878,Z 73,A 1.6589,B 24.8838,C -2.4884,E1 25.1584,E2 82.4699} C_DIS
LIN {X 65.2478,Y 5.2065,Z 73,A -1.7156,B 24.8838,C -2.4889,E1 25.1594,E2 85.8232} C_DIS
LIN {X 65.4498,Y 0.8808,Z 73,A -5.8379,B 24.8856,C -2.4683,E1 25.1598,E2 89.9696} C_DIS
LIN {X 65.3619,Y -3.496,Z 73,A -9.9879,B 24.8875,C -2.448,E1 25.1594,E2 94.143} C_DIS
LIN {X 64.9703,Y -7.9601,Z 73,A -13.6049,B 24.8879,C -2.4434,E1 25.1583,E2 97.7493} C_DIS
LIN {X 64.4266,Y -11.5587,Z 73,A -17.6123,B 24.8908,C -2.4122,E1 25.1564,E2 101.8069} C_DIS
LIN {X 63.6135,Y -15.418,Z 73,A -19.4972,B 24.8881,C -2.442,E1 25.1553,E2 103.6107} C_DIS
LIN {X 62.7183,Y -18.7296,Z 73,A -22.8078,B 24.8897,C -2.4246,E1 25.1528,E2 106.9434} C_DIS
LIN {X 62.1951,Y -20.4017,Z 73,A -25.3804,B 24.8925,C -2.393,E1 25.1505,E2 109.576} C_DIS
LIN {X 61.0033,Y -23.7284,Z 73,A -27.5474,B 24.8912,C -2.4075,E1 25.1484,E2 111.6967} C_DIS
LIN {X 60.3287,Y -25.3936,Z 73,A -29.6651,B 24.8929,C -2.3887,E1 25.146,E2 113.8472} C_DIS
Enddeposition()
END
